LIN {X 0,Y 489.087,Z 544.467,A -85,B 0,C 180,E1 9559.123,E2 9559.123} C_VEL
LIN {X 0,Y 482.604,Z 533.679,A -85,B 0,C 180,E1 9556.552,E2 9556.552} C_VEL
LIN {X 0,Y 477.311,Z 525.25,A -85,B 0,C 180,E1 9554.126,E2 9554.126} C_VEL
LIN {X 0,Y 472.627,Z 517.972,A -85,B 0,C 180,E1 9551.594,E2 9551.594} C_VEL
LIN {X 0,Y 468.762,Z 512.462,A -85,B 0,C 180,E1 9549.082,E2 9549.082} C_VEL
LIN {X 0,Y 465.949,Z 508.396,A -85,B 0,C 180,E1 9546.778,E2 9546.778} C_VEL
LIN {X 0,Y 462.714,Z 503.783,A -85,B 0,C 180,E1 9542.973,E2 9542.973} C_VEL
LIN {X 0,Y 461.058,Z 502.625,A -85,B 0,C 180,E1 9538.633,E2 9538.633} C_VEL
LIN {X 0,Y 461.515,Z 503.464,A -85,B 0,C 180,E1 9534.904,E2 9534.904} C_VEL
LIN {X 0,Y 464.15,Z 508.528,A -85,B 0,C 180,E1 9530.452,E2 9530.452} C_VEL
LIN {X 0,Y 466.705,Z 513.105,A -85,B 0,C 180,E1 9527.943,E2 9527.943} C_VEL
LIN {X 0,Y 469.386,Z 517.69,A -85,B 0,C 180,E1 9525.883,E2 9525.883} C_VEL
LIN {X 0,Y 473.496,Z 524.733,A -85,B 0,C 180,E1 9523.31,E2 9523.31} C_VEL
LIN {X 0,Y 478.239,Z 533.162,A -85,B 0,C 180,E1 9520.837,E2 9520.837} C_VEL
LIN {X 0,Y 483.823,Z 543.406,A -85,B 0,C 180,E1 9518.352,E2 9518.352} C_VEL
LIN {X 0,Y 486.849,Z 549.446,A -85,B 0,C 180,E1 9517.13,E2 9517.13} C_VEL
LIN {X 0,Y 469.793,Z 770.047,A -85,B 0,C 180,E1 9513.766,E2 9513.766} C_VEL
LIN {X 0,Y 464.867,Z 832.514,A -85,B 0,C 180,E1 9512.789,E2 9512.789} C_VEL
LIN {X 0,Y 461.013,Z 860.821,A -85,B 0,C 180,E1 9512.23,E2 9512.23} C_VEL
LIN {X 0,Y 456.896,Z 882.855,A -85,B 0,C 180,E1 9511.67,E2 9511.67} C_VEL
LIN {X 0,Y 452.009,Z 904.689,A -85,B 0,C 180,E1 9510.965,E2 9510.965} C_VEL
LIN {X 0,Y 444.928,Z 930.987,A -85,B 0,C 180,E1 9509.906,E2 9509.906} C_VEL
LIN {X 0,Y 438.503,Z 951.402,A -85,B 0,C 180,E1 9508.895,E2 9508.895} C_VEL
LIN {X 0,Y 431.873,Z 970.249,A -85,B 0,C 180,E1 9507.802,E2 9507.802} C_VEL
LIN {X 0,Y 424.141,Z 990.229,A -85,B 0,C 180,E1 9506.445,E2 9506.445} C_VEL
LIN {X 0,Y 414.213,Z 1013.37,A -85,B 0,C 180,E1 9504.558,E2 9504.558} C_VEL
LIN {X 0,Y 405.888,Z 1031.129,A -85,B 0,C 180,E1 9502.837,E2 9502.837} C_VEL
LIN {X 0,Y 397.662,Z 1047.641,A -85,B 0,C 180,E1 9500.982,E2 9500.982} C_VEL
LIN {X 0,Y 387.672,Z 1066.656,A -85,B 0,C 180,E1 9498.481,E2 9498.481} C_VEL
LIN {X 0,Y 378.087,Z 1083.695,A -85,B 0,C 180,E1 9495.781,E2 9495.781} C_VEL
LIN {X 0,Y 370.336,Z 1097.136,A -85,B 0,C 180,E1 9493.297,E2 9493.297} C_VEL
LIN {X 0,Y 362.061,Z 1111.27,A -85,B 0,C 180,E1 9490.258,E2 9490.258} C_VEL
LIN {X 0,Y 353.591,Z 1125.519,A -85,B 0,C 180,E1 9486.572,E2 9486.572} C_VEL
LIN {X 0,Y 347.43,Z 1136.024,A -85,B 0,C 180,E1 9483.346,E2 9483.346} C_VEL
LIN {X 0,Y 342.159,Z 1145.378,A -85,B 0,C 180,E1 9479.981,E2 9479.981} C_VEL
LIN {X 0,Y 336.708,Z 1155.721,A -85,B 0,C 180,E1 9475.505,E2 9475.505} C_VEL
LIN {X 0,Y 333.16,Z 1163.164,A -85,B 0,C 180,E1 9471.478,E2 9471.478} C_VEL
LIN {X 0,Y 330.879,Z 1168.771,A -85,B 0,C 180,E1 9467.771,E2 9467.771} C_VEL
LIN {X 0,Y 329.229,Z 1173.859,A -85,B 0,C 180,E1 9463.524,E2 9463.524} C_VEL
LIN {X 0,Y 328.351,Z 1177.679,A -85,B 0,C 180,E1 9458.935,E2 9458.935} C_VEL
LIN {X 0,Y 328.063,Z 1179.621,A -85,B 0,C 180,E1 9455.247,E2 9455.247} C_VEL
LIN {X 0,Y 327.994,Z 1180.54,A -85,B 0,C 180,E1 9451.747,E2 9451.747} C_VEL
LIN {X 0,Y 327.999,Z 1180.575,A -85,B 0,C 180,E1 9448.428,E2 9448.428} C_VEL
LIN {X 0,Y 328.045,Z 1179.79,A -85,B 0,C 180,E1 9445.105,E2 9445.105} C_VEL
LIN {X 0,Y 328.254,Z 1178.177,A -85,B 0,C 180,E1 9441.769,E2 9441.769} C_VEL
LIN {X 0,Y 328.768,Z 1175.569,A -85,B 0,C 180,E1 9438.243,E2 9438.243} C_VEL
LIN {X 0,Y 329.903,Z 1171.61,A -85,B 0,C 180,E1 9434.351,E2 9434.351} C_VEL
LIN {X 0,Y 332.358,Z 1165.084,A -85,B 0,C 180,E1 9429.576,E2 9429.576} C_VEL
LIN {X 0,Y 335.423,Z 1158.303,A -85,B 0,C 180,E1 9425.709,E2 9425.709} C_VEL
LIN {X 0,Y 339.344,Z 1150.606,A -85,B 0,C 180,E1 9422.064,E2 9422.064} C_VEL
LIN {X 0,Y 345.374,Z 1139.797,A -85,B 0,C 180,E1 9417.813,E2 9417.813} C_VEL
LIN {X 0,Y 352.237,Z 1127.86,A -85,B 0,C 180,E1 9414.001,E2 9414.001} C_VEL
LIN {X 0,Y 358.846,Z 1116.71,A -85,B 0,C 180,E1 9410.971,E2 9410.971} C_VEL
LIN {X 0,Y 367.61,Z 1102.065,A -85,B 0,C 180,E1 9407.582,E2 9407.582} C_VEL
LIN {X 0,Y 368.215,Z 1100.984,A -85,B 0,C 180,E1 9407.364,E2 9407.364} C_VEL
LIN {X 0,Y 369.925,Z 1096.753,A -85,B 0,C 180,E1 9406.396,E2 9406.396} C_VEL
LIN {X 0,Y 371.745,Z 1086.41,A -85,B 0,C 180,E1 9403.741,E2 9403.741} C_VEL
LIN {X 0,Y 373.805,Z 1081.808,A -85,B 0,C 180,E1 9402.827,E2 9402.827} C_VEL
LIN {X 0,Y 384.889,Z 1062.383,A -85,B 0,C 180,E1 9399.856,E2 9399.856} C_VEL
LIN {X 0,Y 393.525,Z 1046.374,A -85,B 0,C 180,E1 9397.797,E2 9397.797} C_VEL
LIN {X 0,Y 402.328,Z 1029.123,A -85,B 0,C 180,E1 9395.887,E2 9395.887} C_VEL
LIN {X 0,Y 413.045,Z 1006.428,A -85,B 0,C 180,E1 9393.779,E2 9393.779} C_VEL
LIN {X 0,Y 421.336,Z 987.025,A -85,B 0,C 180,E1 9392.273,E2 9392.273} C_VEL
LIN {X 0,Y 428.705,Z 968.221,A -85,B 0,C 180,E1 9391.028,E2 9391.028} C_VEL
LIN {X 0,Y 436.952,Z 944.961,A -85,B 0,C 180,E1 9389.726,E2 9389.726} C_VEL
LIN {X 0,Y 444.264,Z 920.669,A -85,B 0,C 180,E1 9388.629,E2 9388.629} C_VEL
LIN {X 0,Y 449.42,Z 901.022,A -85,B 0,C 180,E1 9387.895,E2 9387.895} C_VEL
LIN {X 0,Y 454.189,Z 879.65,A -85,B 0,C 180,E1 9387.232,E2 9387.232} C_VEL
LIN {X 0,Y 459.09,Z 852.254,A -85,B 0,C 180,E1 9386.579,E2 9386.579} C_VEL
LIN {X 0,Y 462.064,Z 828.163,A -85,B 0,C 180,E1 9386.14,E2 9386.14} C_VEL
LIN {X 0,Y 479.945,Z 602.016,A -85,B 0,C 180,E1 9382.681,E2 9382.681} C_VEL
LIN {X 0,Y 483.792,Z 554.098,A -85,B 0,C 180,E1 9381.936,E2 9381.936} C_VEL
LIN {X 0,Y 478.876,Z 544.784,A -85,B 0,C 180,E1 9379.802,E2 9379.802} C_VEL
LIN {X 0,Y 473.793,Z 535.388,A -85,B 0,C 180,E1 9377.248,E2 9377.248} C_VEL
LIN {X 0,Y 469.705,Z 528.051,A -85,B 0,C 180,E1 9374.8,E2 9374.8} C_VEL
LIN {X 0,Y 466.764,Z 522.997,A -85,B 0,C 180,E1 9372.684,E2 9372.684} C_VEL
LIN {X 0,Y 464.505,Z 518.955,A -85,B 0,C 180,E1 9370.668,E2 9370.668} C_VEL
LIN {X 0,Y 462.693,Z 515.548,A -85,B 0,C 180,E1 9368.575,E2 9368.575} C_VEL
LIN {X 0,Y 460.581,Z 511.278,A -85,B 0,C 180,E1 9364.233,E2 9364.233} C_VEL
LIN {X 0,Y 460.586,Z 510.886,A -85,B 0,C 180,E1 9360.124,E2 9360.124} C_VEL
LIN {X 0,Y 462.046,Z 512.115,A -85,B 0,C 180,E1 9356.899,E2 9356.899} C_VEL
LIN {X 0,Y 465.598,Z 517.283,A -85,B 0,C 180,E1 9352.813,E2 9352.813} C_VEL
LIN {X 0,Y 468.807,Z 522.051,A -85,B 0,C 180,E1 9350.3,E2 9350.3} C_VEL
LIN {X 0,Y 472.497,Z 527.678,A -85,B 0,C 180,E1 9347.969,E2 9347.969} C_VEL
LIN {X 0,Y 476.763,Z 534.255,A -85,B 0,C 180,E1 9345.703,E2 9345.703} C_VEL
LIN {X 0,Y 482.388,Z 543.628,A -85,B 0,C 180,E1 9343.131,E2 9343.131} C_VEL
LIN {X 0,Y 485.974,Z 549.849,A -85,B 0,C 180,E1 9341.67,E2 9341.67} C_VEL
LIN {X 0,Y 467.737,Z 771.285,A -85,B 0,C 180,E1 9338.178,E2 9338.178} C_VEL
LIN {X 0,Y 462.75,Z 830.028,A -85,B 0,C 180,E1 9337.224,E2 9337.224} C_VEL
LIN {X 0,Y 458.58,Z 859.423,A -85,B 0,C 180,E1 9336.635,E2 9336.635} C_VEL
LIN {X 0,Y 454.315,Z 881.758,A -85,B 0,C 180,E1 9336.059,E2 9336.059} C_VEL
LIN {X 0,Y 449.542,Z 902.729,A -85,B 0,C 180,E1 9335.387,E2 9335.387} C_VEL
LIN {X 0,Y 443.382,Z 925.948,A -85,B 0,C 180,E1 9334.486,E2 9334.486} C_VEL
LIN {X 0,Y 435.171,Z 952.253,A -85,B 0,C 180,E1 9333.221,E2 9333.221} C_VEL
LIN {X 0,Y 427.918,Z 972.779,A -85,B 0,C 180,E1 9332.035,E2 9332.035} C_VEL
LIN {X 0,Y 420.219,Z 992.621,A -85,B 0,C 180,E1 9330.695,E2 9330.695} C_VEL
LIN {X 0,Y 410.557,Z 1015.499,A -85,B 0,C 180,E1 9328.875,E2 9328.875} C_VEL
LIN {X 0,Y 400.827,Z 1036.337,A -85,B 0,C 180,E1 9326.886,E2 9326.886} C_VEL
LIN {X 0,Y 392.615,Z 1052.989,A -85,B 0,C 180,E1 9325.039,E2 9325.039} C_VEL
LIN {X 0,Y 384.33,Z 1068.988,A -85,B 0,C 180,E1 9323.005,E2 9323.005} C_VEL
LIN {X 0,Y 374.751,Z 1086.828,A -85,B 0,C 180,E1 9320.38,E2 9320.38} C_VEL
LIN {X 0,Y 364.261,Z 1105.498,A -85,B 0,C 180,E1 9317.097,E2 9317.097} C_VEL
LIN {X 0,Y 356.529,Z 1119.082,A -85,B 0,C 180,E1 9314.291,E2 9314.291} C_VEL
LIN {X 0,Y 349.143,Z 1132.063,A -85,B 0,C 180,E1 9311.198,E2 9311.198} C_VEL
LIN {X 0,Y 341.061,Z 1146.648,A -85,B 0,C 180,E1 9307.115,E2 9307.115} C_VEL
LIN {X 0,Y 334.709,Z 1158.415,A -85,B 0,C 180,E1 9303.139,E2 9303.139} C_VEL
LIN {X 0,Y 330.228,Z 1167.436,A -85,B 0,C 180,E1 9299.573,E2 9299.573} C_VEL
LIN {X 0,Y 326.523,Z 1175.647,A -85,B 0,C 180,E1 9295.774,E2 9295.774} C_VEL
LIN {X 0,Y 323.261,Z 1184.188,A -85,B 0,C 180,E1 9291.026,E2 9291.026} C_VEL
LIN {X 0,Y 321.327,Z 1190.525,A -85,B 0,C 180,E1 9286.449,E2 9286.449} C_VEL
LIN {X 0,Y 320.465,Z 1194.51,A -85,B 0,C 180,E1 9282.798,E2 9282.798} C_VEL
LIN {X 0,Y 320.083,Z 1197.498,A -85,B 0,C 180,E1 9279.167,E2 9279.167} C_VEL
LIN {X 0,Y 319.974,Z 1199.429,A -85,B 0,C 180,E1 9275.739,E2 9275.739} C_VEL
LIN {X 0,Y 319.968,Z 1200.477,A -85,B 0,C 180,E1 9272.328,E2 9272.328} C_VEL
LIN {X 0,Y 319.971,Z 1200.644,A -85,B 0,C 180,E1 9268.925,E2 9268.925} C_VEL
LIN {X 0,Y 319.965,Z 1199.856,A -85,B 0,C 180,E1 9265.339,E2 9265.339} C_VEL
LIN {X 0,Y 320.041,Z 1198.091,A -85,B 0,C 180,E1 9261.737,E2 9261.737} C_VEL
LIN {X 0,Y 320.327,Z 1195.341,A -85,B 0,C 180,E1 9258.111,E2 9258.111} C_VEL
LIN {X 0,Y 321.061,Z 1191.597,A -85,B 0,C 180,E1 9254.464,E2 9254.464} C_VEL
LIN {X 0,Y 322.419,Z 1186.569,A -85,B 0,C 180,E1 9250.62,E2 9250.62} C_VEL
LIN {X 0,Y 324.462,Z 1180.714,A -85,B 0,C 180,E1 9246.96,E2 9246.96} C_VEL
LIN {X 0,Y 327.643,Z 1173.043,A -85,B 0,C 180,E1 9242.954,E2 9242.954} C_VEL
LIN {X 0,Y 333.044,Z 1161.711,A -85,B 0,C 180,E1 9238.103,E2 9238.103} C_VEL
LIN {X 0,Y 338.43,Z 1151.31,A -85,B 0,C 180,E1 9234.406,E2 9234.406} C_VEL
LIN {X 0,Y 344.378,Z 1140.469,A -85,B 0,C 180,E1 9231.09,E2 9231.09} C_VEL
LIN {X 0,Y 351.395,Z 1128.08,A -85,B 0,C 180,E1 9227.815,E2 9227.815} C_VEL
LIN {X 0,Y 361.198,Z 1110.841,A -85,B 0,C 180,E1 9223.967,E2 9223.967} C_VEL
LIN {X 0,Y 369.441,Z 1096.146,A -85,B 0,C 180,E1 9221.201,E2 9221.201} C_VEL
LIN {X 0,Y 377.651,Z 1081.262,A -85,B 0,C 180,E1 9218.773,E2 9218.773} C_VEL
LIN {X 0,Y 386.777,Z 1064.204,A -85,B 0,C 180,E1 9216.363,E2 9216.363} C_VEL
LIN {X 0,Y 397.957,Z 1042.084,A -85,B 0,C 180,E1 9213.73,E2 9213.73} C_VEL
LIN {X 0,Y 406.908,Z 1023.145,A -85,B 0,C 180,E1 9211.835,E2 9211.835} C_VEL
LIN {X 0,Y 415.23,Z 1004.37,A -85,B 0,C 180,E1 9210.217,E2 9210.217} C_VEL
LIN {X 0,Y 424.56,Z 981.647,A -85,B 0,C 180,E1 9208.544,E2 9208.544} C_VEL
LIN {X 0,Y 433.034,Z 958.176,A -85,B 0,C 180,E1 9207.111,E2 9207.111} C_VEL
LIN {X 0,Y 439.667,Z 937.838,A -85,B 0,C 180,E1 9206.064,E2 9206.064} C_VEL
LIN {X 0,Y 445.723,Z 916.98,A -85,B 0,C 180,E1 9205.155,E2 9205.155} C_VEL
LIN {X 0,Y 452.319,Z 890.732,A -85,B 0,C 180,E1 9204.217,E2 9204.217} C_VEL
LIN {X 0,Y 457.368,Z 865.454,A -85,B 0,C 180,E1 9203.515,E2 9203.515} C_VEL
LIN {X 0,Y 460.917,Z 843.374,A -85,B 0,C 180,E1 9203.034,E2 9203.034} C_VEL
LIN {X 0,Y 463.734,Z 818.818,A -85,B 0,C 180,E1 9202.591,E2 9202.591} C_VEL
LIN {X 0,Y 481.973,Z 595.843,A -85,B 0,C 180,E1 9199.059,E2 9199.059} C_VEL
LIN {X 0,Y 485.822,Z 549.536,A -85,B 0,C 180,E1 9198.324,E2 9198.324} C_VEL
LIN {X 0,Y 478.853,Z 537.763,A -85,B 0,C 180,E1 9195.378,E2 9195.378} C_VEL
LIN {X 0,Y 473.264,Z 528.913,A -85,B 0,C 180,E1 9192.569,E2 9192.569} C_VEL
LIN {X 0,Y 470.141,Z 524.264,A -85,B 0,C 180,E1 9190.725,E2 9190.725} C_VEL
LIN {X 0,Y 467.433,Z 520.15,A -85,B 0,C 180,E1 9188.86,E2 9188.86} C_VEL
LIN {X 0,Y 464.829,Z 516.268,A -85,B 0,C 180,E1 9186.671,E2 9186.671} C_VEL
LIN {X 0,Y 461.652,Z 511.681,A -85,B 0,C 180,E1 9182.855,E2 9182.855} C_VEL
LIN {X 0,Y 460.081,Z 510.564,A -85,B 0,C 180,E1 9178.607,E2 9178.607} C_VEL
LIN {X 0,Y 460.501,Z 511.348,A -85,B 0,C 180,E1 9175.017,E2 9175.017} C_VEL
LIN {X 0,Y 463.017,Z 516.34,A -85,B 0,C 180,E1 9170.616,E2 9170.616} C_VEL
LIN {X 0,Y 465.518,Z 520.942,A -85,B 0,C 180,E1 9168.1,E2 9168.1} C_VEL
LIN {X 0,Y 468.15,Z 525.563,A -85,B 0,C 180,E1 9166.034,E2 9166.034} C_VEL
LIN {X 0,Y 471.989,Z 532.31,A -85,B 0,C 180,E1 9163.572,E2 9163.572} C_VEL
LIN {X 0,Y 476.548,Z 540.594,A -85,B 0,C 180,E1 9161.134,E2 9161.134} C_VEL
LIN {X 0,Y 481.912,Z 550.674,A -85,B 0,C 180,E1 9158.685,E2 9158.685} C_VEL
LIN {X 0,Y 483.658,Z 554.297,A -85,B 0,C 180,E1 9157.946,E2 9157.946} C_VEL
LIN {X 0,Y 466.085,Z 776.087,A -85,B 0,C 180,E1 9154.572,E2 9154.572} C_VEL
LIN {X 0,Y 461.441,Z 833.039,A -85,B 0,C 180,E1 9153.681,E2 9153.681} C_VEL
LIN {X 0,Y 457.508,Z 861.097,A -85,B 0,C 180,E1 9153.129,E2 9153.129} C_VEL
LIN {X 0,Y 453.293,Z 883.182,A -85,B 0,C 180,E1 9152.571,E2 9152.571} C_VEL
LIN {X 0,Y 448.197,Z 905.439,A -85,B 0,C 180,E1 9151.856,E2 9151.856} C_VEL
LIN {X 0,Y 440.972,Z 931.565,A -85,B 0,C 180,E1 9150.805,E2 9150.805} C_VEL
LIN {X 0,Y 434.412,Z 951.92,A -85,B 0,C 180,E1 9149.801,E2 9149.801} C_VEL
LIN {X 0,Y 427.637,Z 970.722,A -85,B 0,C 180,E1 9148.715,E2 9148.715} C_VEL
LIN {X 0,Y 419.173,Z 992.057,A -85,B 0,C 180,E1 9147.262,E2 9147.262} C_VEL
LIN {X 0,Y 409.25,Z 1014.406,A -85,B 0,C 180,E1 9145.423,E2 9145.423} C_VEL
LIN {X 0,Y 400.725,Z 1032.084,A -85,B 0,C 180,E1 9143.702,E2 9143.702} C_VEL
LIN {X 0,Y 392.007,Z 1049.072,A -85,B 0,C 180,E1 9141.777,E2 9141.777} C_VEL
LIN {X 0,Y 381.06,Z 1069.057,A -85,B 0,C 180,E1 9139.086,E2 9139.086} C_VEL
LIN {X 0,Y 372.4,Z 1083.999,A -85,B 0,C 180,E1 9136.688,E2 9136.688} C_VEL
LIN {X 0,Y 363.931,Z 1098.184,A -85,B 0,C 180,E1 9134.036,E2 9134.036} C_VEL
LIN {X 0,Y 354.599,Z 1113.556,A -85,B 0,C 180,E1 9130.645,E2 9130.645} C_VEL
LIN {X 0,Y 346.39,Z 1126.747,A -85,B 0,C 180,E1 9127.106,E2 9127.106} C_VEL
LIN {X 0,Y 339.955,Z 1137.294,A -85,B 0,C 180,E1 9123.772,E2 9123.772} C_VEL
LIN {X 0,Y 333.509,Z 1148.386,A -85,B 0,C 180,E1 9119.605,E2 9119.605} C_VEL
LIN {X 0,Y 328.4,Z 1157.61,A -85,B 0,C 180,E1 9115.272,E2 9115.272} C_VEL
LIN {X 0,Y 325.124,Z 1164.296,A -85,B 0,C 180,E1 9111.468,E2 9111.468} C_VEL
LIN {X 0,Y 322.483,Z 1170.734,A -85,B 0,C 180,E1 9106.945,E2 9106.945} C_VEL
LIN {X 0,Y 320.934,Z 1175.425,A -85,B 0,C 180,E1 9102.414,E2 9102.414} C_VEL
LIN {X 0,Y 320.322,Z 1178.252,A -85,B 0,C 180,E1 9098.618,E2 9098.618} C_VEL
LIN {X 0,Y 320.057,Z 1179.998,A -85,B 0,C 180,E1 9095.019,E2 9095.019} C_VEL
LIN {X 0,Y 319.997,Z 1180.809,A -85,B 0,C 180,E1 9091.612,E2 9091.612} C_VEL
LIN {X 0,Y 320.006,Z 1180.8,A -85,B 0,C 180,E1 9088.21,E2 9088.21} C_VEL
LIN {X 0,Y 320.062,Z 1179.973,A -85,B 0,C 180,E1 9084.802,E2 9084.802} C_VEL
LIN {X 0,Y 320.332,Z 1178.21,A -85,B 0,C 180,E1 9081.203,E2 9081.203} C_VEL
LIN {X 0,Y 321.004,Z 1175.212,A -85,B 0,C 180,E1 9077.224,E2 9077.224} C_VEL
LIN {X 0,Y 322.785,Z 1169.902,A -85,B 0,C 180,E1 9072.328,E2 9072.328} C_VEL
LIN {X 0,Y 325.195,Z 1164.177,A -85,B 0,C 180,E1 9068.349,E2 9068.349} C_VEL
LIN {X 0,Y 328.462,Z 1157.543,A -85,B 0,C 180,E1 9064.582,E2 9064.582} C_VEL
LIN {X 0,Y 333.698,Z 1148.116,A -85,B 0,C 180,E1 9060.173,E2 9060.173} C_VEL
LIN {X 0,Y 340.123,Z 1137.072,A -85,B 0,C 180,E1 9056.045,E2 9056.045} C_VEL
LIN {X 0,Y 346.595,Z 1126.496,A -85,B 0,C 180,E1 9052.713,E2 9052.713} C_VEL
LIN {X 0,Y 355.244,Z 1112.617,A -85,B 0,C 180,E1 9049.02,E2 9049.02} C_VEL
LIN {X 0,Y 364.316,Z 1097.665,A -85,B 0,C 180,E1 9045.753,E2 9045.753} C_VEL
LIN {X 0,Y 372.539,Z 1083.908,A -85,B 0,C 180,E1 9043.19,E2 9043.19} C_VEL
LIN {X 0,Y 373.805,Z 1081.808,A -85,B 0,C 180,E1 9042.827,E2 9042.827} C_VEL
LIN {X 0,Y 375.924,Z 1077.178,A -85,B 0,C 180,E1 9041.932,E2 9041.932} C_VEL
LIN {X 0,Y 378.862,Z 1065.068,A -85,B 0,C 180,E1 9039.326,E2 9039.326} C_VEL
LIN {X 0,Y 380.839,Z 1060.662,A -85,B 0,C 180,E1 9038.629,E2 9038.629} C_VEL
LIN {X 0,Y 389.359,Z 1045.266,A -85,B 0,C 180,E1 9036.675,E2 9036.675} C_VEL
LIN {X 0,Y 398.942,Z 1026.928,A -85,B 0,C 180,E1 9034.677,E2 9034.677} C_VEL
LIN {X 0,Y 409.366,Z 1005.103,A -85,B 0,C 180,E1 9032.695,E2 9032.695} C_VEL
LIN {X 0,Y 417.191,Z 987.19,A -85,B 0,C 180,E1 9031.318,E2 9031.318} C_VEL
LIN {X 0,Y 424.767,Z 968.28,A -85,B 0,C 180,E1 9030.072,E2 9030.072} C_VEL
LIN {X 0,Y 433.029,Z 945.469,A -85,B 0,C 180,E1 9028.804,E2 9028.804} C_VEL
LIN {X 0,Y 440.491,Z 921.305,A -85,B 0,C 180,E1 9027.716,E2 9027.716} C_VEL
LIN {X 0,Y 445.748,Z 901.755,A -85,B 0,C 180,E1 9026.99,E2 9026.99} C_VEL
LIN {X 0,Y 450.512,Z 880.944,A -85,B 0,C 180,E1 9026.344,E2 9026.344} C_VEL
LIN {X 0,Y 455.419,Z 854.865,A -85,B 0,C 180,E1 9025.713,E2 9025.713} C_VEL
LIN {X 0,Y 458.75,Z 828.848,A -85,B 0,C 180,E1 9025.237,E2 9025.237} C_VEL
LIN {X 0,Y 477.095,Z 602.943,A -85,B 0,C 180,E1 9021.793,E2 9021.793} C_VEL
LIN {X 0,Y 480.703,Z 559.088,A -85,B 0,C 180,E1 9021.112,E2 9021.112} C_VEL
LIN {X 0,Y 475.753,Z 549.457,A -85,B 0,C 180,E1 9018.821,E2 9018.821} C_VEL
LIN {X 0,Y 471.327,Z 541.288,A -85,B 0,C 180,E1 9016.452,E2 9016.452} C_VEL
LIN {X 0,Y 467.998,Z 535.179,A -85,B 0,C 180,E1 9014.35,E2 9014.35} C_VEL
LIN {X 0,Y 465.483,Z 530.695,A -85,B 0,C 180,E1 9012.467,E2 9012.467} C_VEL
LIN {X 0,Y 463.167,Z 526.461,A -85,B 0,C 180,E1 9010.322,E2 9010.322} C_VEL
LIN {X 0,Y 461.534,Z 523.318,A -85,B 0,C 180,E1 9008.346,E2 9008.346} C_VEL
LIN {X 0,Y 459.608,Z 519.226,A -85,B 0,C 180,E1 9004.242,E2 9004.242} C_VEL
LIN {X 0,Y 459.58,Z 518.808,A -85,B 0,C 180,E1 9000.249,E2 9000.249} C_VEL
LIN {X 0,Y 461.055,Z 520.15,A -85,B 0,C 180,E1 8996.892,E2 8996.892} C_VEL
LIN {X 0,Y 464.429,Z 525.143,A -85,B 0,C 180,E1 8992.951,E2 8992.951} C_VEL
LIN {X 0,Y 467.545,Z 529.883,A -85,B 0,C 180,E1 8990.46,E2 8990.46} C_VEL
LIN {X 0,Y 470.977,Z 535.209,A -85,B 0,C 180,E1 8988.24,E2 8988.24} C_VEL
LIN {X 0,Y 475.148,Z 541.808,A -85,B 0,C 180,E1 8985.964,E2 8985.964} C_VEL
LIN {X 0,Y 480.604,Z 551.1,A -85,B 0,C 180,E1 8983.408,E2 8983.408} C_VEL
LIN {X 0,Y 482.79,Z 555.033,A -85,B 0,C 180,E1 8982.482,E2 8982.482} C_VEL
LIN {X 0,Y 464.15,Z 776.331,A -85,B 0,C 180,E1 8979.005,E2 8979.005} C_VEL
LIN {X 0,Y 459.389,Z 830.749,A -85,B 0,C 180,E1 8978.122,E2 8978.122} C_VEL
LIN {X 0,Y 455.185,Z 859.62,A -85,B 0,C 180,E1 8977.546,E2 8977.546} C_VEL
LIN {X 0,Y 450.857,Z 881.859,A -85,B 0,C 180,E1 8976.977,E2 8976.977} C_VEL
LIN {X 0,Y 445.848,Z 903.395,A -85,B 0,C 180,E1 8976.292,E2 8976.292} C_VEL
LIN {X 0,Y 439.052,Z 928.394,A -85,B 0,C 180,E1 8975.321,E2 8975.321} C_VEL
LIN {X 0,Y 431.135,Z 952.846,A -85,B 0,C 180,E1 8974.136,E2 8974.136} C_VEL
LIN {X 0,Y 423.86,Z 972.947,A -85,B 0,C 180,E1 8972.98,E2 8972.98} C_VEL
LIN {X 0,Y 415.898,Z 992.984,A -85,B 0,C 180,E1 8971.631,E2 8971.631} C_VEL
LIN {X 0,Y 405.668,Z 1016.473,A -85,B 0,C 180,E1 8969.757,E2 8969.757} C_VEL
LIN {X 0,Y 395.819,Z 1036.987,A -85,B 0,C 180,E1 8967.791,E2 8967.791} C_VEL
LIN {X 0,Y 387.347,Z 1053.65,A -85,B 0,C 180,E1 8965.933,E2 8965.933} C_VEL
LIN {X 0,Y 378.44,Z 1070.303,A -85,B 0,C 180,E1 8963.795,E2 8963.795} C_VEL
LIN {X 0,Y 367.511,Z 1089.864,A -85,B 0,C 180,E1 8960.84,E2 8960.84} C_VEL
LIN {X 0,Y 358.041,Z 1106.068,A -85,B 0,C 180,E1 8957.914,E2 8957.914} C_VEL
LIN {X 0,Y 350.099,Z 1119.505,A -85,B 0,C 180,E1 8955.095,E2 8955.095} C_VEL
LIN {X 0,Y 342.062,Z 1133.078,A -85,B 0,C 180,E1 8951.794,E2 8951.794} C_VEL
LIN {X 0,Y 333.141,Z 1148.406,A -85,B 0,C 180,E1 8947.32,E2 8947.32} C_VEL
LIN {X 0,Y 327.417,Z 1158.614,A -85,B 0,C 180,E1 8943.765,E2 8943.765} C_VEL
LIN {X 0,Y 322.731,Z 1167.585,A -85,B 0,C 180,E1 8940.126,E2 8940.126} C_VEL
LIN {X 0,Y 318.692,Z 1176.115,A -85,B 0,C 180,E1 8936.055,E2 8936.055} C_VEL
LIN {X 0,Y 315.112,Z 1184.993,A -85,B 0,C 180,E1 8930.817,E2 8930.817} C_VEL
LIN {X 0,Y 313.388,Z 1190.485,A -85,B 0,C 180,E1 8926.687,E2 8926.687} C_VEL
LIN {X 0,Y 312.484,Z 1194.425,A -85,B 0,C 180,E1 8922.943,E2 8922.943} C_VEL
LIN {X 0,Y 312.093,Z 1197.297,A -85,B 0,C 180,E1 8919.326,E2 8919.326} C_VEL
LIN {X 0,Y 311.977,Z 1199.18,A -85,B 0,C 180,E1 8915.886,E2 8915.886} C_VEL
LIN {X 0,Y 311.971,Z 1200.23,A -85,B 0,C 180,E1 8912.388,E2 8912.388} C_VEL
LIN {X 0,Y 311.975,Z 1200.397,A -85,B 0,C 180,E1 8908.898,E2 8908.898} C_VEL
LIN {X 0,Y 311.969,Z 1199.608,A -85,B 0,C 180,E1 8905.22,E2 8905.22} C_VEL
LIN {X 0,Y 312.049,Z 1197.84,A -85,B 0,C 180,E1 8901.524,E2 8901.524} C_VEL
LIN {X 0,Y 312.368,Z 1195.087,A -85,B 0,C 180,E1 8897.803,E2 8897.803} C_VEL
LIN {X 0,Y 313.162,Z 1191.339,A -85,B 0,C 180,E1 8894.062,E2 8894.062} C_VEL
LIN {X 0,Y 314.595,Z 1186.399,A -85,B 0,C 180,E1 8890.185,E2 8890.185} C_VEL
LIN {X 0,Y 316.816,Z 1180.448,A -85,B 0,C 180,E1 8886.371,E2 8886.371} C_VEL
LIN {X 0,Y 320.383,Z 1172.405,A -85,B 0,C 180,E1 8882.086,E2 8882.086} C_VEL
LIN {X 0,Y 326.157,Z 1160.955,A -85,B 0,C 180,E1 8877.138,E2 8877.138} C_VEL
LIN {X 0,Y 331.9,Z 1150.493,A -85,B 0,C 180,E1 8873.38,E2 8873.38} C_VEL
LIN {X 0,Y 338.363,Z 1139.315,A -85,B 0,C 180,E1 8869.94,E2 8869.94} C_VEL
LIN {X 0,Y 347.169,Z 1124.474,A -85,B 0,C 180,E1 8866.044,E2 8866.044} C_VEL
LIN {X 0,Y 356.28,Z 1108.946,A -85,B 0,C 180,E1 8862.668,E2 8862.668} C_VEL
LIN {X 0,Y 364.431,Z 1094.959,A -85,B 0,C 180,E1 8860.05,E2 8860.05} C_VEL
LIN {X 0,Y 373.255,Z 1079.477,A -85,B 0,C 180,E1 8857.54,E2 8857.54} C_VEL
LIN {X 0,Y 384.164,Z 1059.637,A -85,B 0,C 180,E1 8854.798,E2 8854.798} C_VEL
LIN {X 0,Y 394.283,Z 1039.864,A -85,B 0,C 180,E1 8852.522,E2 8852.522} C_VEL
LIN {X 0,Y 403.035,Z 1021.759,A -85,B 0,C 180,E1 8850.735,E2 8850.735} C_VEL
LIN {X 0,Y 412.535,Z 1000.739,A -85,B 0,C 180,E1 8848.958,E2 8848.958} C_VEL
LIN {X 0,Y 422.368,Z 976.596,A -85,B 0,C 180,E1 8847.261,E2 8847.261} C_VEL
LIN {X 0,Y 429.696,Z 956.617,A -85,B 0,C 180,E1 8846.077,E2 8846.077} C_VEL
LIN {X 0,Y 436.122,Z 937.241,A -85,B 0,C 180,E1 8845.095,E2 8845.095} C_VEL
LIN {X 0,Y 442.674,Z 915.012,A -85,B 0,C 180,E1 8844.143,E2 8844.143} C_VEL
LIN {X 0,Y 449.683,Z 886.727,A -85,B 0,C 180,E1 8843.174,E2 8843.174} C_VEL
LIN {X 0,Y 454.204,Z 864.236,A -85,B 0,C 180,E1 8842.569,E2 8842.569} C_VEL
LIN {X 0,Y 457.768,Z 842.166,A -85,B 0,C 180,E1 8842.099,E2 8842.099} C_VEL
LIN {X 0,Y 460.875,Z 814.57,A -85,B 0,C 180,E1 8841.61,E2 8841.61} C_VEL
LIN {X 0,Y 479.731,Z 588.85,A -85,B 0,C 180,E1 8838.053,E2 8838.053} C_VEL
LIN {X 0,Y 482.639,Z 554.74,A -85,B 0,C 180,E1 8837.517,E2 8837.517} C_VEL
LIN {X 0,Y 476.697,Z 544.545,A -85,B 0,C 180,E1 8834.889,E2 8834.889} C_VEL
LIN {X 0,Y 471.612,Z 536.292,A -85,B 0,C 180,E1 8832.241,E2 8832.241} C_VEL
LIN {X 0,Y 468.577,Z 531.674,A -85,B 0,C 180,E1 8830.388,E2 8830.388} C_VEL
LIN {X 0,Y 466.113,Z 527.837,A -85,B 0,C 180,E1 8828.636,E2 8828.636} C_VEL
LIN {X 0,Y 463.577,Z 524.003,A -85,B 0,C 180,E1 8826.44,E2 8826.44} C_VEL
LIN {X 0,Y 460.591,Z 519.579,A -85,B 0,C 180,E1 8822.737,E2 8822.737} C_VEL
LIN {X 0,Y 459.097,Z 518.501,A -85,B 0,C 180,E1 8818.502,E2 8818.502} C_VEL
LIN {X 0,Y 459.52,Z 519.366,A -85,B 0,C 180,E1 8815.007,E2 8815.007} C_VEL
LIN {X 0,Y 461.887,Z 524.151,A -85,B 0,C 180,E1 8810.782,E2 8810.782} C_VEL
LIN {X 0,Y 464.328,Z 528.776,A -85,B 0,C 180,E1 8808.258,E2 8808.258} C_VEL
LIN {X 0,Y 466.753,Z 533.117,A -85,B 0,C 180,E1 8806.307,E2 8806.307} C_VEL
LIN {X 0,Y 470.429,Z 539.755,A -85,B 0,C 180,E1 8803.874,E2 8803.874} C_VEL
LIN {X 0,Y 474.879,Z 548.036,A -85,B 0,C 180,E1 8801.43,E2 8801.43} C_VEL
LIN {X 0,Y 479.982,Z 557.868,A -85,B 0,C 180,E1 8799.036,E2 8799.036} C_VEL
LIN {X 0,Y 480.559,Z 559.318,A -85,B 0,C 180,E1 8798.77,E2 8798.77} C_VEL
LIN {X 0,Y 462.56,Z 781.004,A -85,B 0,C 180,E1 8795.409,E2 8795.409} C_VEL
LIN {X 0,Y 458.095,Z 833.883,A -85,B 0,C 180,E1 8794.581,E2 8794.581} C_VEL
LIN {X 0,Y 454.115,Z 861.388,A -85,B 0,C 180,E1 8794.04,E2 8794.04} C_VEL
LIN {X 0,Y 449.827,Z 883.404,A -85,B 0,C 180,E1 8793.489,E2 8793.489} C_VEL
LIN {X 0,Y 444.677,Z 905.455,A -85,B 0,C 180,E1 8792.786,E2 8792.786} C_VEL
LIN {X 0,Y 437.126,Z 932.142,A -85,B 0,C 180,E1 8791.721,E2 8791.721} C_VEL
LIN {X 0,Y 430.432,Z 952.438,A -85,B 0,C 180,E1 8790.724,E2 8790.724} C_VEL
LIN {X 0,Y 423.589,Z 970.993,A -85,B 0,C 180,E1 8789.658,E2 8789.658} C_VEL
LIN {X 0,Y 414.734,Z 992.801,A -85,B 0,C 180,E1 8788.178,E2 8788.178} C_VEL
LIN {X 0,Y 404.702,Z 1014.784,A -85,B 0,C 180,E1 8786.368,E2 8786.368} C_VEL
LIN {X 0,Y 395.964,Z 1032.443,A -85,B 0,C 180,E1 8784.65,E2 8784.65} C_VEL
LIN {X 0,Y 386.728,Z 1049.944,A -85,B 0,C 180,E1 8782.662,E2 8782.662} C_VEL
LIN {X 0,Y 375.198,Z 1070.276,A -85,B 0,C 180,E1 8779.893,E2 8779.893} C_VEL
LIN {X 0,Y 366.304,Z 1085.131,A -85,B 0,C 180,E1 8777.477,E2 8777.477} C_VEL
LIN {X 0,Y 357.13,Z 1099.986,A -85,B 0,C 180,E1 8774.648,E2 8774.648} C_VEL
LIN {X 0,Y 346.895,Z 1116.053,A -85,B 0,C 180,E1 8770.958,E2 8770.958} C_VEL
LIN {X 0,Y 339.473,Z 1127.582,A -85,B 0,C 180,E1 8767.781,E2 8767.781} C_VEL
LIN {X 0,Y 332.805,Z 1138.067,A -85,B 0,C 180,E1 8764.391,E2 8764.391} C_VEL
LIN {X 0,Y 325.66,Z 1149.736,A -85,B 0,C 180,E1 8759.828,E2 8759.828} C_VEL
LIN {X 0,Y 320.804,Z 1158.17,A -85,B 0,C 180,E1 8755.741,E2 8755.741} C_VEL
LIN {X 0,Y 317.36,Z 1164.848,A -85,B 0,C 180,E1 8751.825,E2 8751.825} C_VEL
LIN {X 0,Y 314.506,Z 1171.411,A -85,B 0,C 180,E1 8747.007,E2 8747.007} C_VEL
LIN {X 0,Y 312.972,Z 1175.828,A -85,B 0,C 180,E1 8742.548,E2 8742.548} C_VEL
LIN {X 0,Y 312.332,Z 1178.609,A -85,B 0,C 180,E1 8738.654,E2 8738.654} C_VEL
LIN {X 0,Y 312.06,Z 1180.311,A -85,B 0,C 180,E1 8734.963,E2 8734.963} C_VEL
LIN {X 0,Y 312.003,Z 1181.099,A -85,B 0,C 180,E1 8731.286,E2 8731.286} C_VEL
LIN {X 0,Y 312.012,Z 1180.984,A -85,B 0,C 180,E1 8727.613,E2 8727.613} C_VEL
LIN {X 0,Y 312.161,Z 1179.709,A -85,B 0,C 180,E1 8723.194,E2 8723.194} C_VEL
LIN {X 0,Y 312.715,Z 1176.831,A -85,B 0,C 180,E1 8718.566,E2 8718.566} C_VEL
LIN {X 0,Y 313.86,Z 1173.103,A -85,B 0,C 180,E1 8714.479,E2 8714.479} C_VEL
LIN {X 0,Y 315.708,Z 1168.452,A -85,B 0,C 180,E1 8710.577,E2 8710.577} C_VEL
LIN {X 0,Y 319.102,Z 1161.523,A -85,B 0,C 180,E1 8705.962,E2 8705.962} C_VEL
LIN {X 0,Y 323.928,Z 1152.697,A -85,B 0,C 180,E1 8701.417,E2 8701.417} C_VEL
LIN {X 0,Y 328.901,Z 1144.386,A -85,B 0,C 180,E1 8697.859,E2 8697.859} C_VEL
LIN {X 0,Y 335.563,Z 1133.842,A -85,B 0,C 180,E1 8694.056,E2 8694.056} C_VEL
LIN {X 0,Y 344.183,Z 1120.358,A -85,B 0,C 180,E1 8690.058,E2 8690.058} C_VEL
LIN {X 0,Y 352.022,Z 1108.116,A -85,B 0,C 180,E1 8687.025,E2 8687.025} C_VEL
LIN {X 0,Y 360.246,Z 1095.118,A -85,B 0,C 180,E1 8684.268,E2 8684.268} C_VEL
LIN {X 0,Y 370.775,Z 1078.016,A -85,B 0,C 180,E1 8681.203,E2 8681.203} C_VEL
LIN {X 0,Y 380.839,Z 1060.662,A -85,B 0,C 180,E1 8678.629,E2 8678.629} C_VEL
LIN {X 0,Y 383.13,Z 1055.589,A -85,B 0,C 180,E1 8677.819,E2 8677.819} C_VEL
LIN {X 0,Y 386.851,Z 1042.392,A -85,B 0,C 180,E1 8675.402,E2 8675.402} C_VEL
LIN {X 0,Y 388.916,Z 1037.652,A -85,B 0,C 180,E1 8674.785,E2 8674.785} C_VEL
LIN {X 0,Y 398.767,Z 1018.463,A -85,B 0,C 180,E1 8672.862,E2 8672.862} C_VEL
LIN {X 0,Y 407.34,Z 1000.495,A -85,B 0,C 180,E1 8671.327,E2 8671.327} C_VEL
LIN {X 0,Y 416.662,Z 979.252,A -85,B 0,C 180,E1 8669.785,E2 8669.785} C_VEL
LIN {X 0,Y 425.654,Z 955.915,A -85,B 0,C 180,E1 8668.393,E2 8668.393} C_VEL
LIN {X 0,Y 432.091,Z 937.166,A -85,B 0,C 180,E1 8667.448,E2 8667.448} C_VEL
LIN {X 0,Y 438.286,Z 916.844,A -85,B 0,C 180,E1 8666.584,E2 8666.584} C_VEL
LIN {X 0,Y 444.795,Z 892.188,A -85,B 0,C 180,E1 8665.729,E2 8665.729} C_VEL
LIN {X 0,Y 450.121,Z 866.522,A -85,B 0,C 180,E1 8665.047,E2 8665.047} C_VEL
LIN {X 0,Y 453.639,Z 844.978,A -85,B 0,C 180,E1 8664.596,E2 8664.596} C_VEL
LIN {X 0,Y 456.508,Z 820.105,A -85,B 0,C 180,E1 8664.168,E2 8664.168} C_VEL
LIN {X 0,Y 475.434,Z 591.235,A -85,B 0,C 180,E1 8660.702,E2 8660.702} C_VEL
LIN {X 0,Y 477.688,Z 564.063,A -85,B 0,C 180,E1 8660.269,E2 8660.269} C_VEL
LIN {X 0,Y 472.35,Z 553.588,A -85,B 0,C 180,E1 8657.62,E2 8657.62} C_VEL
LIN {X 0,Y 467.644,Z 544.664,A -85,B 0,C 180,E1 8654.804,E2 8654.804} C_VEL
LIN {X 0,Y 464.283,Z 538.514,A -85,B 0,C 180,E1 8652.311,E2 8652.311} C_VEL
LIN {X 0,Y 461.959,Z 534.167,A -85,B 0,C 180,E1 8650.097,E2 8650.097} C_VEL
LIN {X 0,Y 460.474,Z 531.201,A -85,B 0,C 180,E1 8648.24,E2 8648.24} C_VEL
LIN {X 0,Y 458.602,Z 527.135,A -85,B 0,C 180,E1 8644.126,E2 8644.126} C_VEL
LIN {X 0,Y 458.636,Z 526.77,A -85,B 0,C 180,E1 8640.125,E2 8640.125} C_VEL
LIN {X 0,Y 459.996,Z 528.027,A -85,B 0,C 180,E1 8637.01,E2 8637.01} C_VEL
LIN {X 0,Y 463.231,Z 532.943,A -85,B 0,C 180,E1 8633.12,E2 8633.12} C_VEL
LIN {X 0,Y 466.207,Z 537.565,A -85,B 0,C 180,E1 8630.681,E2 8630.681} C_VEL
LIN {X 0,Y 469.663,Z 543.057,A -85,B 0,C 180,E1 8628.394,E2 8628.394} C_VEL
LIN {X 0,Y 473.769,Z 549.769,A -85,B 0,C 180,E1 8626.109,E2 8626.109} C_VEL
LIN {X 0,Y 479.097,Z 559.029,A -85,B 0,C 180,E1 8623.573,E2 8623.573} C_VEL
LIN {X 0,Y 479.685,Z 560.327,A -85,B 0,C 180,E1 8623.303,E2 8623.303} C_VEL
LIN {X 0,Y 460.709,Z 780.763,A -85,B 0,C 180,E1 8619.854,E2 8619.854} C_VEL
LIN {X 0,Y 456.147,Z 831.439,A -85,B 0,C 180,E1 8619.033,E2 8619.033} C_VEL
LIN {X 0,Y 451.898,Z 859.876,A -85,B 0,C 180,E1 8618.468,E2 8618.468} C_VEL
LIN {X 0,Y 447.517,Z 881.963,A -85,B 0,C 180,E1 8617.909,E2 8617.909} C_VEL
LIN {X 0,Y 442.417,Z 903.466,A -85,B 0,C 180,E1 8617.233,E2 8617.233} C_VEL
LIN {X 0,Y 435.322,Z 929.001,A -85,B 0,C 180,E1 8616.248,E2 8616.248} C_VEL
LIN {X 0,Y 427.247,Z 953.341,A -85,B 0,C 180,E1 8615.074,E2 8615.074} C_VEL
LIN {X 0,Y 420.071,Z 972.733,A -85,B 0,C 180,E1 8613.967,E2 8613.967} C_VEL
LIN {X 0,Y 412.03,Z 992.542,A -85,B 0,C 180,E1 8612.644,E2 8612.644} C_VEL
LIN {X 0,Y 401.886,Z 1015.41,A -85,B 0,C 180,E1 8610.841,E2 8610.841} C_VEL
LIN {X 0,Y 391.471,Z 1036.559,A -85,B 0,C 180,E1 8608.83,E2 8608.83} C_VEL
LIN {X 0,Y 382.768,Z 1053.202,A -85,B 0,C 180,E1 8606.984,E2 8606.984} C_VEL
LIN {X 0,Y 373.724,Z 1069.618,A -85,B 0,C 180,E1 8604.884,E2 8604.884} C_VEL
LIN {X 0,Y 362.782,Z 1088.688,A -85,B 0,C 180,E1 8602.022,E2 8602.022} C_VEL
LIN {X 0,Y 352.56,Z 1105.568,A -85,B 0,C 180,E1 8598.971,E2 8598.971} C_VEL
LIN {X 0,Y 344.187,Z 1119.209,A -85,B 0,C 180,E1 8596.091,E2 8596.091} C_VEL
LIN {X 0,Y 336.201,Z 1132.135,A -85,B 0,C 180,E1 8592.926,E2 8592.926} C_VEL
LIN {X 0,Y 327.106,Z 1147.061,A -85,B 0,C 180,E1 8588.577,E2 8588.577} C_VEL
LIN {X 0,Y 320.443,Z 1158.34,A -85,B 0,C 180,E1 8584.603,E2 8584.603} C_VEL
LIN {X 0,Y 315.481,Z 1167.313,A -85,B 0,C 180,E1 8580.893,E2 8580.893} C_VEL
LIN {X 0,Y 311.183,Z 1175.883,A -85,B 0,C 180,E1 8576.713,E2 8576.713} C_VEL
LIN {X 0,Y 307.379,Z 1184.733,A -85,B 0,C 180,E1 8571.366,E2 8571.366} C_VEL
LIN {X 0,Y 305.51,Z 1190.237,A -85,B 0,C 180,E1 8567.122,E2 8567.122} C_VEL
LIN {X 0,Y 304.539,Z 1194.172,A -85,B 0,C 180,E1 8563.286,E2 8563.286} C_VEL
LIN {X 0,Y 304.101,Z 1197.12,A -85,B 0,C 180,E1 8559.457,E2 8559.457} C_VEL
LIN {X 0,Y 303.979,Z 1199.004,A -85,B 0,C 180,E1 8555.852,E2 8555.852} C_VEL
LIN {X 0,Y 303.974,Z 1200.007,A -85,B 0,C 180,E1 8552.262,E2 8552.262} C_VEL
LIN {X 0,Y 303.979,Z 1200.126,A -85,B 0,C 180,E1 8548.68,E2 8548.68} C_VEL
LIN {X 0,Y 303.972,Z 1199.359,A -85,B 0,C 180,E1 8545.093,E2 8545.093} C_VEL
LIN {X 0,Y 304.059,Z 1197.589,A -85,B 0,C 180,E1 8541.299,E2 8541.299} C_VEL
LIN {X 0,Y 304.416,Z 1194.833,A -85,B 0,C 180,E1 8537.48,E2 8537.48} C_VEL
LIN {X 0,Y 305.274,Z 1191.081,A -85,B 0,C 180,E1 8533.639,E2 8533.639} C_VEL
LIN {X 0,Y 306.762,Z 1186.311,A -85,B 0,C 180,E1 8529.787,E2 8529.787} C_VEL
LIN {X 0,Y 309.064,Z 1180.498,A -85,B 0,C 180,E1 8525.943,E2 8525.943} C_VEL
LIN {X 0,Y 312.427,Z 1173.239,A -85,B 0,C 180,E1 8521.936,E2 8521.936} C_VEL
LIN {X 0,Y 317.853,Z 1163.052,A -85,B 0,C 180,E1 8517.243,E2 8517.243} C_VEL
LIN {X 0,Y 324.53,Z 1151.274,A -85,B 0,C 180,E1 8512.852,E2 8512.852} C_VEL
LIN {X 0,Y 330.912,Z 1140.678,A -85,B 0,C 180,E1 8509.485,E2 8509.485} C_VEL
LIN {X 0,Y 338.21,Z 1128.798,A -85,B 0,C 180,E1 8506.227,E2 8506.227} C_VEL
LIN {X 0,Y 347.803,Z 1113.365,A -85,B 0,C 180,E1 8502.611,E2 8502.611} C_VEL
LIN {X 0,Y 358.029,Z 1096.373,A -85,B 0,C 180,E1 8499.323,E2 8499.323} C_VEL
LIN {X 0,Y 367.076,Z 1081.044,A -85,B 0,C 180,E1 8496.791,E2 8496.791} C_VEL
LIN {X 0,Y 376.402,Z 1064.671,A -85,B 0,C 180,E1 8494.46,E2 8494.46} C_VEL
LIN {X 0,Y 388.291,Z 1042.58,A -85,B 0,C 180,E1 8491.812,E2 8491.812} C_VEL
LIN {X 0,Y 397.882,Z 1023.356,A -85,B 0,C 180,E1 8489.889,E2 8489.889} C_VEL
LIN {X 0,Y 406.542,Z 1004.8,A -85,B 0,C 180,E1 8488.298,E2 8488.298} C_VEL
LIN {X 0,Y 415.824,Z 983.299,A -85,B 0,C 180,E1 8486.722,E2 8486.722} C_VEL
LIN {X 0,Y 425.06,Z 959.137,A -85,B 0,C 180,E1 8485.248,E2 8485.248} C_VEL
LIN {X 0,Y 431.969,Z 938.934,A -85,B 0,C 180,E1 8484.218,E2 8484.218} C_VEL
LIN {X 0,Y 438.264,Z 918.235,A -85,B 0,C 180,E1 8483.323,E2 8483.323} C_VEL
LIN {X 0,Y 444.488,Z 894.769,A -85,B 0,C 180,E1 8482.484,E2 8482.484} C_VEL
LIN {X 0,Y 450.397,Z 867.205,A -85,B 0,C 180,E1 8481.71,E2 8481.71} C_VEL
LIN {X 0,Y 454.194,Z 844.708,A -85,B 0,C 180,E1 8481.224,E2 8481.224} C_VEL
LIN {X 0,Y 456.989,Z 821.922,A -85,B 0,C 180,E1 8480.813,E2 8480.813} C_VEL
LIN {X 0,Y 475.518,Z 606.098,A -85,B 0,C 180,E1 8477.415,E2 8477.415} C_VEL
LIN {X 0,Y 479.538,Z 559.935,A -85,B 0,C 180,E1 8476.692,E2 8476.692} C_VEL
LIN {X 0,Y 473.825,Z 550.031,A -85,B 0,C 180,E1 8474.014,E2 8474.014} C_VEL
LIN {X 0,Y 469.671,Z 543.203,A -85,B 0,C 180,E1 8471.731,E2 8471.731} C_VEL
LIN {X 0,Y 466.852,Z 538.805,A -85,B 0,C 180,E1 8469.928,E2 8469.928} C_VEL
LIN {X 0,Y 464.801,Z 535.525,A -85,B 0,C 180,E1 8468.412,E2 8468.412} C_VEL
LIN {X 0,Y 462.458,Z 531.876,A -85,B 0,C 180,E1 8466.331,E2 8466.331} C_VEL
LIN {X 0,Y 459.533,Z 527.477,A -85,B 0,C 180,E1 8462.619,E2 8462.619} C_VEL
LIN {X 0,Y 458.116,Z 526.441,A -85,B 0,C 180,E1 8458.434,E2 8458.434} C_VEL
LIN {X 0,Y 458.507,Z 527.25,A -85,B 0,C 180,E1 8455.121,E2 8455.121} C_VEL
LIN {X 0,Y 460.809,Z 532.07,A -85,B 0,C 180,E1 8450.886,E2 8450.886} C_VEL
LIN {X 0,Y 463.142,Z 536.609,A -85,B 0,C 180,E1 8448.417,E2 8448.417} C_VEL
LIN {X 0,Y 465.527,Z 540.987,A -85,B 0,C 180,E1 8446.46,E2 8446.46} C_VEL
LIN {X 0,Y 469.008,Z 547.457,A -85,B 0,C 180,E1 8444.1,E2 8444.1} C_VEL
LIN {X 0,Y 473.305,Z 555.637,A -85,B 0,C 180,E1 8441.685,E2 8441.685} C_VEL
LIN {X 0,Y 477.578,Z 564.101,A -85,B 0,C 180,E1 8439.608,E2 8439.608} C_VEL
LIN {X 0,Y 459.122,Z 785.976,A -85,B 0,C 180,E1 8436.256,E2 8436.256} C_VEL
LIN {X 0,Y 454.854,Z 834.824,A -85,B 0,C 180,E1 8435.492,E2 8435.492} C_VEL
LIN {X 0,Y 450.839,Z 861.677,A -85,B 0,C 180,E1 8434.965,E2 8434.965} C_VEL
LIN {X 0,Y 446.472,Z 883.651,A -85,B 0,C 180,E1 8434.42,E2 8434.42} C_VEL
LIN {X 0,Y 441.09,Z 906.201,A -85,B 0,C 180,E1 8433.706,E2 8433.706} C_VEL
LIN {X 0,Y 433.393,Z 932.716,A -85,B 0,C 180,E1 8432.652,E2 8432.652} C_VEL
LIN {X 0,Y 426.921,Z 951.962,A -85,B 0,C 180,E1 8431.717,E2 8431.717} C_VEL
LIN {X 0,Y 419.849,Z 970.776,A -85,B 0,C 180,E1 8430.65,E2 8430.65} C_VEL
LIN {X 0,Y 410.912,Z 992.333,A -85,B 0,C 180,E1 8429.2,E2 8429.2} C_VEL
LIN {X 0,Y 400.375,Z 1014.941,A -85,B 0,C 180,E1 8427.355,E2 8427.355} C_VEL
LIN {X 0,Y 391.63,Z 1032.199,A -85,B 0,C 180,E1 8425.684,E2 8425.684} C_VEL
LIN {X 0,Y 382.566,Z 1048.957,A -85,B 0,C 180,E1 8423.794,E2 8423.794} C_VEL
LIN {X 0,Y 371.1,Z 1068.771,A -85,B 0,C 180,E1 8421.139,E2 8421.139} C_VEL
LIN {X 0,Y 361.327,Z 1084.603,A -85,B 0,C 180,E1 8418.584,E2 8418.584} C_VEL
LIN {X 0,Y 352.536,Z 1098.366,A -85,B 0,C 180,E1 8415.981,E2 8415.981} C_VEL
LIN {X 0,Y 342.666,Z 1113.492,A -85,B 0,C 180,E1 8412.607,E2 8412.607} C_VEL
LIN {X 0,Y 333.728,Z 1126.741,A -85,B 0,C 180,E1 8408.99,E2 8408.99} C_VEL
LIN {X 0,Y 326.669,Z 1137.34,A -85,B 0,C 180,E1 8405.561,E2 8405.561} C_VEL
LIN {X 0,Y 319.575,Z 1148.406,A -85,B 0,C 180,E1 8401.291,E2 8401.291} C_VEL
LIN {X 0,Y 313.733,Z 1157.866,A -85,B 0,C 180,E1 8396.704,E2 8396.704} C_VEL
LIN {X 0,Y 310.005,Z 1164.612,A -85,B 0,C 180,E1 8392.71,E2 8392.71} C_VEL
LIN {X 0,Y 307.088,Z 1170.76,A -85,B 0,C 180,E1 8388.215,E2 8388.215} C_VEL
LIN {X 0,Y 305.162,Z 1175.777,A -85,B 0,C 180,E1 8383.26,E2 8383.26} C_VEL
LIN {X 0,Y 304.386,Z 1178.751,A -85,B 0,C 180,E1 8379.072,E2 8379.072} C_VEL
LIN {X 0,Y 304.079,Z 1180.494,A -85,B 0,C 180,E1 8375.283,E2 8375.283} C_VEL
LIN {X 0,Y 304.005,Z 1181.303,A -85,B 0,C 180,E1 8371.697,E2 8371.697} C_VEL
LIN {X 0,Y 304.013,Z 1181.294,A -85,B 0,C 180,E1 8368.116,E2 8368.116} C_VEL
LIN {X 0,Y 304.084,Z 1180.469,A -85,B 0,C 180,E1 8364.529,E2 8364.529} C_VEL
LIN {X 0,Y 304.395,Z 1178.708,A -85,B 0,C 180,E1 8360.738,E2 8360.738} C_VEL
LIN {X 0,Y 305.196,Z 1175.714,A -85,B 0,C 180,E1 8356.55,E2 8356.55} C_VEL
LIN {X 0,Y 307.24,Z 1170.412,A -85,B 0,C 180,E1 8351.402,E2 8351.402} C_VEL
LIN {X 0,Y 310.131,Z 1164.401,A -85,B 0,C 180,E1 8347.039,E2 8347.039} C_VEL
LIN {X 0,Y 313.846,Z 1157.722,A -85,B 0,C 180,E1 8343.103,E2 8343.103} C_VEL
LIN {X 0,Y 319.729,Z 1148.207,A -85,B 0,C 180,E1 8338.517,E2 8338.517} C_VEL
LIN {X 0,Y 326.536,Z 1137.609,A -85,B 0,C 180,E1 8334.424,E2 8334.424} C_VEL
LIN {X 0,Y 333.584,Z 1127.04,A -85,B 0,C 180,E1 8330.991,E2 8330.991} C_VEL
LIN {X 0,Y 342.939,Z 1113.184,A -85,B 0,C 180,E1 8327.209,E2 8327.209} C_VEL
LIN {X 0,Y 352.582,Z 1098.421,A -85,B 0,C 180,E1 8323.92,E2 8323.92} C_VEL
LIN {X 0,Y 361.147,Z 1085.04,A -85,B 0,C 180,E1 8321.385,E2 8321.385} C_VEL
LIN {X 0,Y 370.909,Z 1069.242,A -85,B 0,C 180,E1 8318.825,E2 8318.825} C_VEL
LIN {X 0,Y 382.534,Z 1049.22,A -85,B 0,C 180,E1 8316.132,E2 8316.132} C_VEL
LIN {X 0,Y 388.916,Z 1037.652,A -85,B 0,C 180,E1 8314.785,E2 8314.785} C_VEL
LIN {X 0,Y 391.241,Z 1032.161,A -85,B 0,C 180,E1 8314.071,E2 8314.071} C_VEL
LIN {X 0,Y 395.046,Z 1018.616,A -85,B 0,C 180,E1 8311.974,E2 8311.974} C_VEL
LIN {X 0,Y 397.53,Z 1012.721,A -85,B 0,C 180,E1 8311.321,E2 8311.321} C_VEL
LIN {X 0,Y 408.025,Z 990.356,A -85,B 0,C 180,E1 8309.549,E2 8309.549} C_VEL
LIN {X 0,Y 416.481,Z 970.325,A -85,B 0,C 180,E1 8308.227,E2 8308.227} C_VEL
LIN {X 0,Y 424.068,Z 950.449,A -85,B 0,C 180,E1 8307.118,E2 8307.118} C_VEL
LIN {X 0,Y 432.189,Z 926.385,A -85,B 0,C 180,E1 8306,E2 8306} C_VEL
LIN {X 0,Y 438.743,Z 903.205,A -85,B 0,C 180,E1 8305.135,E2 8305.135} C_VEL
LIN {X 0,Y 443.754,Z 882.326,A -85,B 0,C 180,E1 8304.494,E2 8304.494} C_VEL
LIN {X 0,Y 448.368,Z 859.14,A -85,B 0,C 180,E1 8303.933,E2 8303.933} C_VEL
LIN {X 0,Y 452.406,Z 830.867,A -85,B 0,C 180,E1 8303.405,E2 8303.405} C_VEL
LIN {X 0,Y 459.979,Z 742.643,A -85,B 0,C 180,E1 8302.055,E2 8302.055} C_VEL
LIN {X 0,Y 474.821,Z 569.132,A -85,B 0,C 180,E1 8299.434,E2 8299.434} C_VEL
LIN {X 0,Y 469.363,Z 558.26,A -85,B 0,C 180,E1 8296.529,E2 8296.529} C_VEL
LIN {X 0,Y 465.432,Z 550.728,A -85,B 0,C 180,E1 8293.986,E2 8293.986} C_VEL
LIN {X 0,Y 462.8,Z 545.847,A -85,B 0,C 180,E1 8291.907,E2 8291.907} C_VEL
LIN {X 0,Y 460.75,Z 541.858,A -85,B 0,C 180,E1 8289.862,E2 8289.862} C_VEL
LIN {X 0,Y 459.326,Z 538.969,A -85,B 0,C 180,E1 8288.009,E2 8288.009} C_VEL
LIN {X 0,Y 457.598,Z 535.044,A -85,B 0,C 180,E1 8284.01,E2 8284.01} C_VEL
LIN {X 0,Y 457.659,Z 534.711,A -85,B 0,C 180,E1 8280.125,E2 8280.125} C_VEL
LIN {X 0,Y 458.938,Z 535.905,A -85,B 0,C 180,E1 8277.128,E2 8277.128} C_VEL
LIN {X 0,Y 462.038,Z 540.741,A -85,B 0,C 180,E1 8273.289,E2 8273.289} C_VEL
LIN {X 0,Y 464.876,Z 545.246,A -85,B 0,C 180,E1 8270.904,E2 8270.904} C_VEL
LIN {X 0,Y 468.254,Z 550.745,A -85,B 0,C 180,E1 8268.608,E2 8268.608} C_VEL
LIN {X 0,Y 472.339,Z 557.618,A -85,B 0,C 180,E1 8266.285,E2 8266.285} C_VEL
LIN {X 0,Y 476.709,Z 565.362,A -85,B 0,C 180,E1 8264.141,E2 8264.141} C_VEL
LIN {X 0,Y 457.615,Z 782.462,A -85,B 0,C 180,E1 8260.759,E2 8260.759} C_VEL
LIN {X 0,Y 453.033,Z 832.033,A -85,B 0,C 180,E1 8259.959,E2 8259.959} C_VEL
LIN {X 0,Y 448.721,Z 860.17,A -85,B 0,C 180,E1 8259.403,E2 8259.403} C_VEL
LIN {X 0,Y 444.298,Z 882.071,A -85,B 0,C 180,E1 8258.855,E2 8258.855} C_VEL
LIN {X 0,Y 439.127,Z 903.465,A -85,B 0,C 180,E1 8258.191,E2 8258.191} C_VEL
LIN {X 0,Y 432.087,Z 928.382,A -85,B 0,C 180,E1 8257.243,E2 8257.243} C_VEL
LIN {X 0,Y 423.846,Z 952.821,A -85,B 0,C 180,E1 8256.082,E2 8256.082} C_VEL
LIN {X 0,Y 416.552,Z 972.166,A -85,B 0,C 180,E1 8254.992,E2 8254.992} C_VEL
LIN {X 0,Y 408.433,Z 991.785,A -85,B 0,C 180,E1 8253.697,E2 8253.697} C_VEL
LIN {X 0,Y 398.587,Z 1013.584,A -85,B 0,C 180,E1 8252.007,E2 8252.007} C_VEL
LIN {X 0,Y 387.691,Z 1035.308,A -85,B 0,C 180,E1 8249.977,E2 8249.977} C_VEL
LIN {X 0,Y 378.559,Z 1052.326,A -85,B 0,C 180,E1 8248.112,E2 8248.112} C_VEL
LIN {X 0,Y 369.397,Z 1068.501,A -85,B 0,C 180,E1 8246.06,E2 8246.06} C_VEL
LIN {X 0,Y 358.2,Z 1087.47,A -85,B 0,C 180,E1 8243.238,E2 8243.238} C_VEL
LIN {X 0,Y 347.074,Z 1105.267,A -85,B 0,C 180,E1 8240.023,E2 8240.023} C_VEL
LIN {X 0,Y 338.375,Z 1118.913,A -85,B 0,C 180,E1 8237.123,E2 8237.123} C_VEL
LIN {X 0,Y 330.059,Z 1131.844,A -85,B 0,C 180,E1 8233.926,E2 8233.926} C_VEL
LIN {X 0,Y 320.529,Z 1146.782,A -85,B 0,C 180,E1 8229.521,E2 8229.521} C_VEL
LIN {X 0,Y 313.541,Z 1158.064,A -85,B 0,C 180,E1 8225.478,E2 8225.478} C_VEL
LIN {X 0,Y 308.291,Z 1167.042,A -85,B 0,C 180,E1 8221.696,E2 8221.696} C_VEL
LIN {X 0,Y 303.744,Z 1175.58,A -85,B 0,C 180,E1 8217.442,E2 8217.442} C_VEL
LIN {X 0,Y 299.659,Z 1184.488,A -85,B 0,C 180,E1 8211.933,E2 8211.933} C_VEL
LIN {X 0,Y 297.649,Z 1189.971,A -85,B 0,C 180,E1 8207.597,E2 8207.597} C_VEL
LIN {X 0,Y 296.6,Z 1193.918,A -85,B 0,C 180,E1 8203.649,E2 8203.649} C_VEL
LIN {X 0,Y 296.119,Z 1196.866,A -85,B 0,C 180,E1 8199.719,E2 8199.719} C_VEL
LIN {X 0,Y 295.983,Z 1198.756,A -85,B 0,C 180,E1 8196.011,E2 8196.011} C_VEL
LIN {X 0,Y 295.977,Z 1199.76,A -85,B 0,C 180,E1 8192.323,E2 8192.323} C_VEL
LIN {X 0,Y 295.983,Z 1199.879,A -85,B 0,C 180,E1 8188.645,E2 8188.645} C_VEL
LIN {X 0,Y 295.975,Z 1199.111,A -85,B 0,C 180,E1 8184.961,E2 8184.961} C_VEL
LIN {X 0,Y 296.072,Z 1197.337,A -85,B 0,C 180,E1 8181.063,E2 8181.063} C_VEL
LIN {X 0,Y 296.474,Z 1194.53,A -85,B 0,C 180,E1 8177.081,E2 8177.081} C_VEL
LIN {X 0,Y 297.399,Z 1190.823,A -85,B 0,C 180,E1 8173.193,E2 8173.193} C_VEL
LIN {X 0,Y 299.011,Z 1186.05,A -85,B 0,C 180,E1 8169.239,E2 8169.239} C_VEL
LIN {X 0,Y 301.469,Z 1180.233,A -85,B 0,C 180,E1 8165.297,E2 8165.297} C_VEL
LIN {X 0,Y 305.054,Z 1172.969,A -85,B 0,C 180,E1 8161.195,E2 8161.195} C_VEL
LIN {X 0,Y 310.791,Z 1162.774,A -85,B 0,C 180,E1 8156.402,E2 8156.402} C_VEL
LIN {X 0,Y 317.842,Z 1150.991,A -85,B 0,C 180,E1 8151.932,E2 8151.932} C_VEL
LIN {X 0,Y 324.898,Z 1139.798,A -85,B 0,C 180,E1 8148.337,E2 8148.337} C_VEL
LIN {X 0,Y 332.993,Z 1127.197,A -85,B 0,C 180,E1 8144.875,E2 8144.875} C_VEL
LIN {X 0,Y 344.065,Z 1109.91,A -85,B 0,C 180,E1 8140.924,E2 8140.924} C_VEL
LIN {X 0,Y 353.365,Z 1095.055,A -85,B 0,C 180,E1 8138.087,E2 8138.087} C_VEL
LIN {X 0,Y 362.736,Z 1079.672,A -85,B 0,C 180,E1 8135.565,E2 8135.565} C_VEL
LIN {X 0,Y 374.122,Z 1060.266,A -85,B 0,C 180,E1 8132.857,E2 8132.857} C_VEL
LIN {X 0,Y 384.922,Z 1040.347,A -85,B 0,C 180,E1 8130.558,E2 8130.558} C_VEL
LIN {X 0,Y 394.135,Z 1022.283,A -85,B 0,C 180,E1 8128.777,E2 8128.777} C_VEL
LIN {X 0,Y 403.38,Z 1002.855,A -85,B 0,C 180,E1 8127.136,E2 8127.136} C_VEL
LIN {X 0,Y 414.34,Z 977.445,A -85,B 0,C 180,E1 8125.346,E2 8125.346} C_VEL
LIN {X 0,Y 422.201,Z 956.98,A -85,B 0,C 180,E1 8124.149,E2 8124.149} C_VEL
LIN {X 0,Y 429.042,Z 937.196,A -85,B 0,C 180,E1 8123.164,E2 8123.164} C_VEL
LIN {X 0,Y 435.72,Z 915.423,A -85,B 0,C 180,E1 8122.25,E2 8122.25} C_VEL
LIN {X 0,Y 443.034,Z 887.092,A -85,B 0,C 180,E1 8121.296,E2 8121.296} C_VEL
LIN {X 0,Y 447.767,Z 864.426,A -85,B 0,C 180,E1 8120.702,E2 8120.702} C_VEL
LIN {X 0,Y 451.455,Z 842.377,A -85,B 0,C 180,E1 8120.241,E2 8120.241} C_VEL
LIN {X 0,Y 454.668,Z 815.021,A -85,B 0,C 180,E1 8119.762,E2 8119.762} C_VEL
LIN {X 0,Y 474.416,Z 589.118,A -85,B 0,C 180,E1 8116.235,E2 8116.235} C_VEL
LIN {X 0,Y 476.517,Z 565.195,A -85,B 0,C 180,E1 8115.851,E2 8115.851} C_VEL
LIN {X 0,Y 471.398,Z 556.061,A -85,B 0,C 180,E1 8113.305,E2 8113.305} C_VEL
LIN {X 0,Y 466.853,Z 548.442,A -85,B 0,C 180,E1 8110.614,E2 8110.614} C_VEL
LIN {X 0,Y 463.497,Z 543.212,A -85,B 0,C 180,E1 8108.186,E2 8108.186} C_VEL
LIN {X 0,Y 461.216,Z 539.608,A -85,B 0,C 180,E1 8106.098,E2 8106.098} C_VEL
LIN {X 0,Y 458.478,Z 535.376,A -85,B 0,C 180,E1 8102.5,E2 8102.5} C_VEL
LIN {X 0,Y 457.147,Z 534.382,A -85,B 0,C 180,E1 8098.496,E2 8098.496} C_VEL
LIN {X 0,Y 457.526,Z 535.274,A -85,B 0,C 180,E1 8095.111,E2 8095.111} C_VEL
LIN {X 0,Y 459.685,Z 539.88,A -85,B 0,C 180,E1 8091.053,E2 8091.053} C_VEL
LIN {X 0,Y 461.894,Z 544.307,A -85,B 0,C 180,E1 8088.639,E2 8088.639} C_VEL
LIN {X 0,Y 464.223,Z 548.698,A -85,B 0,C 180,E1 8086.675,E2 8086.675} C_VEL
LIN {X 0,Y 467.535,Z 555.028,A -85,B 0,C 180,E1 8084.367,E2 8084.367} C_VEL
LIN {X 0,Y 471.683,Z 563.125,A -85,B 0,C 180,E1 8081.971,E2 8081.971} C_VEL
LIN {X 0,Y 474.654,Z 569.348,A -85,B 0,C 180,E1 8080.45,E2 8080.45} C_VEL
LIN {X 0,Y 455.779,Z 791.073,A -85,B 0,C 180,E1 8077.115,E2 8077.115} C_VEL
LIN {X 0,Y 451.659,Z 836.425,A -85,B 0,C 180,E1 8076.405,E2 8076.405} C_VEL
LIN {X 0,Y 447.553,Z 862.662,A -85,B 0,C 180,E1 8075.888,E2 8075.888} C_VEL
LIN {X 0,Y 443.148,Z 884.296,A -85,B 0,C 180,E1 8075.354,E2 8075.354} C_VEL
LIN {X 0,Y 437.242,Z 908.414,A -85,B 0,C 180,E1 8074.593,E2 8074.593} C_VEL
LIN {X 0,Y 429.777,Z 933.289,A -85,B 0,C 180,E1 8073.599,E2 8073.599} C_VEL
LIN {X 0,Y 423.177,Z 952.476,A -85,B 0,C 180,E1 8072.674,E2 8072.674} C_VEL
LIN {X 0,Y 415.964,Z 971.244,A -85,B 0,C 180,E1 8071.616,E2 8071.616} C_VEL
LIN {X 0,Y 406.838,Z 992.766,A -85,B 0,C 180,E1 8070.177,E2 8070.177} C_VEL
LIN {X 0,Y 396.285,Z 1014.876,A -85,B 0,C 180,E1 8068.382,E2 8068.382} C_VEL
LIN {X 0,Y 387.106,Z 1032.553,A -85,B 0,C 180,E1 8066.677,E2 8066.677} C_VEL
LIN {X 0,Y 377.972,Z 1048.998,A -85,B 0,C 180,E1 8064.828,E2 8064.828} C_VEL
LIN {X 0,Y 366.603,Z 1068.173,A -85,B 0,C 180,E1 8062.275,E2 8062.275} C_VEL
LIN {X 0,Y 355.949,Z 1084.905,A -85,B 0,C 180,E1 8059.575,E2 8059.575} C_VEL
LIN {X 0,Y 347.095,Z 1098.313,A -85,B 0,C 180,E1 8057.029,E2 8057.029} C_VEL
LIN {X 0,Y 336.599,Z 1113.823,A -85,B 0,C 180,E1 8053.546,E2 8053.546} C_VEL
LIN {X 0,Y 327.342,Z 1127.017,A -85,B 0,C 180,E1 8049.901,E2 8049.901} C_VEL
LIN {X 0,Y 319.981,Z 1137.61,A -85,B 0,C 180,E1 8046.421,E2 8046.421} C_VEL
LIN {X 0,Y 312.407,Z 1148.885,A -85,B 0,C 180,E1 8041.987,E2 8041.987} C_VEL
LIN {X 0,Y 306.389,Z 1158.129,A -85,B 0,C 180,E1 8037.397,E2 8037.397} C_VEL
LIN {X 0,Y 302.485,Z 1164.783,A -85,B 0,C 180,E1 8033.37,E2 8033.37} C_VEL
LIN {X 0,Y 299.331,Z 1171.017,A -85,B 0,C 180,E1 8028.704,E2 8028.704} C_VEL
LIN {X 0,Y 297.251,Z 1176.077,A -85,B 0,C 180,E1 8023.556,E2 8023.556} C_VEL
LIN {X 0,Y 296.42,Z 1179.002,A -85,B 0,C 180,E1 8019.318,E2 8019.318} C_VEL
LIN {X 0,Y 296.09,Z 1180.743,A -85,B 0,C 180,E1 8015.426,E2 8015.426} C_VEL
LIN {X 0,Y 296.01,Z 1181.55,A -85,B 0,C 180,E1 8011.743,E2 8011.743} C_VEL
LIN {X 0,Y 296.016,Z 1181.563,A -85,B 0,C 180,E1 8008.258,E2 8008.258} C_VEL
LIN {X 0,Y 296.086,Z 1180.781,A -85,B 0,C 180,E1 8004.575,E2 8004.575} C_VEL
LIN {X 0,Y 296.387,Z 1179.173,A -85,B 0,C 180,E1 8000.877,E2 8000.877} C_VEL
LIN {X 0,Y 297.134,Z 1176.421,A -85,B 0,C 180,E1 7996.773,E2 7996.773} C_VEL
LIN {X 0,Y 298.788,Z 1172.228,A -85,B 0,C 180,E1 7992.271,E2 7992.271} C_VEL
LIN {X 0,Y 302.106,Z 1165.532,A -85,B 0,C 180,E1 7987.012,E2 7987.012} C_VEL
LIN {X 0,Y 306.088,Z 1158.661,A -85,B 0,C 180,E1 7982.786,E2 7982.786} C_VEL
LIN {X 0,Y 311.335,Z 1150.48,A -85,B 0,C 180,E1 7978.65,E2 7978.65} C_VEL
LIN {X 0,Y 319.167,Z 1138.877,A -85,B 0,C 180,E1 7973.917,E2 7973.917} C_VEL
LIN {X 0,Y 326.417,Z 1128.427,A -85,B 0,C 180,E1 7970.421,E2 7970.421} C_VEL
LIN {X 0,Y 334.255,Z 1117.197,A -85,B 0,C 180,E1 7967.232,E2 7967.232} C_VEL
LIN {X 0,Y 344.544,Z 1102.335,A -85,B 0,C 180,E1 7963.685,E2 7963.685} C_VEL
LIN {X 0,Y 355.081,Z 1086.39,A -85,B 0,C 180,E1 7960.578,E2 7960.578} C_VEL
LIN {X 0,Y 364.093,Z 1072.272,A -85,B 0,C 180,E1 7958.241,E2 7958.241} C_VEL
LIN {X 0,Y 374.99,Z 1054.423,A -85,B 0,C 180,E1 7955.729,E2 7955.729} C_VEL
LIN {X 0,Y 385.945,Z 1034.955,A -85,B 0,C 180,E1 7953.467,E2 7953.467} C_VEL
LIN {X 0,Y 395.084,Z 1017.513,A -85,B 0,C 180,E1 7951.751,E2 7951.751} C_VEL
LIN {X 0,Y 397.53,Z 1012.721,A -85,B 0,C 180,E1 7951.321,E2 7951.321} C_VEL
LIN {X 0,Y 399.992,Z 1006.826,A -85,B 0,C 180,E1 7950.687,E2 7950.687} C_VEL
LIN {X 0,Y 403.95,Z 992.251,A -85,B 0,C 180,E1 7948.793,E2 7948.793} C_VEL
LIN {X 0,Y 406.225,Z 986.024,A -85,B 0,C 180,E1 7948.227,E2 7948.227} C_VEL
LIN {X 0,Y 414.569,Z 966.331,A -85,B 0,C 180,E1 7946.979,E2 7946.979} C_VEL
LIN {X 0,Y 424.199,Z 940.519,A -85,B 0,C 180,E1 7945.633,E2 7945.633} C_VEL
LIN {X 0,Y 430.994,Z 919.378,A -85,B 0,C 180,E1 7944.736,E2 7944.736} C_VEL
LIN {X 0,Y 436.761,Z 898.79,A -85,B 0,C 180,E1 7944.017,E2 7944.017} C_VEL
LIN {X 0,Y 442.473,Z 874.637,A -85,B 0,C 180,E1 7943.332,E2 7943.332} C_VEL
LIN {X 0,Y 447.157,Z 848.408,A -85,B 0,C 180,E1 7942.766,E2 7942.766} C_VEL
LIN {X 0,Y 450.008,Z 826.195,A -85,B 0,C 180,E1 7942.378,E2 7942.378} C_VEL
LIN {X 0,Y 469.952,Z 597.833,A -85,B 0,C 180,E1 7938.947,E2 7938.947} C_VEL
LIN {X 0,Y 472.024,Z 574.465,A -85,B 0,C 180,E1 7938.591,E2 7938.591} C_VEL
LIN {X 0,Y 467.453,Z 565.085,A -85,B 0,C 180,E1 7936.018,E2 7936.018} C_VEL
LIN {X 0,Y 463.945,Z 558.142,A -85,B 0,C 180,E1 7933.65,E2 7933.65} C_VEL
LIN {X 0,Y 461.475,Z 553.422,A -85,B 0,C 180,E1 7931.625,E2 7931.625} C_VEL
LIN {X 0,Y 459.565,Z 549.578,A -85,B 0,C 180,E1 7929.644,E2 7929.644} C_VEL
LIN {X 0,Y 458.236,Z 546.804,A -85,B 0,C 180,E1 7927.85,E2 7927.85} C_VEL
LIN {X 0,Y 456.624,Z 542.992,A -85,B 0,C 180,E1 7924.018,E2 7924.018} C_VEL
LIN {X 0,Y 456.679,Z 542.652,A -85,B 0,C 180,E1 7920.125,E2 7920.125} C_VEL
LIN {X 0,Y 457.882,Z 543.783,A -85,B 0,C 180,E1 7917.246,E2 7917.246} C_VEL
LIN {X 0,Y 460.909,Z 548.658,A -85,B 0,C 180,E1 7913.398,E2 7913.398} C_VEL
LIN {X 0,Y 463.628,Z 553.074,A -85,B 0,C 180,E1 7911.067,E2 7911.067} C_VEL
LIN {X 0,Y 467.045,Z 558.744,A -85,B 0,C 180,E1 7908.703,E2 7908.703} C_VEL
LIN {X 0,Y 471.764,Z 566.911,A -85,B 0,C 180,E1 7906.018,E2 7906.018} C_VEL
LIN {X 0,Y 473.802,Z 570.875,A -85,B 0,C 180,E1 7904.979,E2 7904.979} C_VEL
LIN {X 0,Y 453.763,Z 794.074,A -85,B 0,C 180,E1 7901.522,E2 7901.522} C_VEL
LIN {X 0,Y 449.708,Z 835.443,A -85,B 0,C 180,E1 7900.849,E2 7900.849} C_VEL
LIN {X 0,Y 445.421,Z 861.755,A -85,B 0,C 180,E1 7900.323,E2 7900.323} C_VEL
LIN {X 0,Y 441.003,Z 883.054,A -85,B 0,C 180,E1 7899.79,E2 7899.79} C_VEL
LIN {X 0,Y 435.574,Z 904.96,A -85,B 0,C 180,E1 7899.112,E2 7899.112} C_VEL
LIN {X 0,Y 427.436,Z 932.424,A -85,B 0,C 180,E1 7898.049,E2 7898.049} C_VEL
LIN {X 0,Y 419.927,Z 954.061,A -85,B 0,C 180,E1 7897.014,E2 7897.014} C_VEL
LIN {X 0,Y 412.356,Z 973.608,A -85,B 0,C 180,E1 7895.913,E2 7895.913} C_VEL
LIN {X 0,Y 403.613,Z 994.138,A -85,B 0,C 180,E1 7894.552,E2 7894.552} C_VEL
LIN {X 0,Y 391.955,Z 1018.72,A -85,B 0,C 180,E1 7892.591,E2 7892.591} C_VEL
LIN {X 0,Y 382.433,Z 1037.073,A -85,B 0,C 180,E1 7890.837,E2 7890.837} C_VEL
LIN {X 0,Y 373.259,Z 1053.641,A -85,B 0,C 180,E1 7889.004,E2 7889.004} C_VEL
LIN {X 0,Y 363.137,Z 1070.955,A -85,B 0,C 180,E1 7886.774,E2 7886.774} C_VEL
LIN {X 0,Y 350.434,Z 1091.461,A -85,B 0,C 180,E1 7883.595,E2 7883.595} C_VEL
LIN {X 0,Y 340.664,Z 1106.545,A -85,B 0,C 180,E1 7880.792,E2 7880.792} C_VEL
LIN {X 0,Y 331.722,Z 1120.058,A -85,B 0,C 180,E1 7877.858,E2 7877.858} C_VEL
LIN {X 0,Y 321.473,Z 1135.435,A -85,B 0,C 180,E1 7873.915,E2 7873.915} C_VEL
LIN {X 0,Y 312.615,Z 1148.633,A -85,B 0,C 180,E1 7869.768,E2 7869.768} C_VEL
LIN {X 0,Y 306.103,Z 1158.742,A -85,B 0,C 180,E1 7866.012,E2 7866.012} C_VEL
LIN {X 0,Y 300.19,Z 1168.453,A -85,B 0,C 180,E1 7861.753,E2 7861.753} C_VEL
LIN {X 0,Y 294.551,Z 1178.732,A -85,B 0,C 180,E1 7856.186,E2 7856.186} C_VEL
LIN {X 0,Y 291.509,Z 1185.279,A -85,B 0,C 180,E1 7851.742,E2 7851.742} C_VEL
LIN {X 0,Y 289.664,Z 1190.149,A -85,B 0,C 180,E1 7847.683,E2 7847.683} C_VEL
LIN {X 0,Y 288.63,Z 1193.833,A -85,B 0,C 180,E1 7843.829,E2 7843.829} C_VEL
LIN {X 0,Y 288.124,Z 1196.736,A -85,B 0,C 180,E1 7839.79,E2 7839.79} C_VEL
LIN {X 0,Y 287.988,Z 1198.507,A -85,B 0,C 180,E1 7836.178,E2 7836.178} C_VEL
LIN {X 0,Y 287.981,Z 1199.488,A -85,B 0,C 180,E1 7832.587,E2 7832.587} C_VEL
LIN {X 0,Y 287.985,Z 1199.655,A -85,B 0,C 180,E1 7828.806,E2 7828.806} C_VEL
LIN {X 0,Y 287.978,Z 1198.862,A -85,B 0,C 180,E1 7824.82,E2 7824.82} C_VEL
LIN {X 0,Y 288.085,Z 1197.086,A -85,B 0,C 180,E1 7820.813,E2 7820.813} C_VEL
LIN {X 0,Y 288.519,Z 1194.324,A -85,B 0,C 180,E1 7816.777,E2 7816.777} C_VEL
LIN {X 0,Y 289.532,Z 1190.565,A -85,B 0,C 180,E1 7812.722,E2 7812.722} C_VEL
LIN {X 0,Y 291.284,Z 1185.789,A -85,B 0,C 180,E1 7808.662,E2 7808.662} C_VEL
LIN {X 0,Y 293.904,Z 1179.967,A -85,B 0,C 180,E1 7804.617,E2 7804.617} C_VEL
LIN {X 0,Y 297.728,Z 1172.701,A -85,B 0,C 180,E1 7800.417,E2 7800.417} C_VEL
LIN {X 0,Y 303.795,Z 1162.496,A -85,B 0,C 180,E1 7795.521,E2 7795.521} C_VEL
LIN {X 0,Y 311.233,Z 1150.709,A -85,B 0,C 180,E1 7790.973,E2 7790.973} C_VEL
LIN {X 0,Y 318.616,Z 1139.511,A -85,B 0,C 180,E1 7787.324,E2 7787.324} C_VEL
LIN {X 0,Y 327.658,Z 1126.06,A -85,B 0,C 180,E1 7783.604,E2 7783.604} C_VEL
LIN {X 0,Y 338.595,Z 1109.603,A -85,B 0,C 180,E1 7779.844,E2 7779.844} C_VEL
LIN {X 0,Y 348.145,Z 1094.876,A -85,B 0,C 180,E1 7777.02,E2 7777.02} C_VEL
LIN {X 0,Y 357.322,Z 1080.291,A -85,B 0,C 180,E1 7774.615,E2 7774.615} C_VEL
LIN {X 0,Y 367.866,Z 1062.848,A -85,B 0,C 180,E1 7772.148,E2 7772.148} C_VEL
LIN {X 0,Y 380.084,Z 1041.217,A -85,B 0,C 180,E1 7769.606,E2 7769.606} C_VEL
LIN {X 0,Y 389.854,Z 1022.572,A -85,B 0,C 180,E1 7767.768,E2 7767.768} C_VEL
LIN {X 0,Y 398.937,Z 1003.966,A -85,B 0,C 180,E1 7766.197,E2 7766.197} C_VEL
LIN {X 0,Y 409.432,Z 980.568,A -85,B 0,C 180,E1 7764.53,E2 7764.53} C_VEL
LIN {X 0,Y 418.303,Z 958.069,A -85,B 0,C 180,E1 7763.208,E2 7763.208} C_VEL
LIN {X 0,Y 425.499,Z 937.749,A -85,B 0,C 180,E1 7762.201,E2 7762.201} C_VEL
LIN {X 0,Y 432.084,Z 916.772,A -85,B 0,C 180,E1 7761.324,E2 7761.324} C_VEL
LIN {X 0,Y 439.245,Z 890.195,A -85,B 0,C 180,E1 7760.422,E2 7760.422} C_VEL
LIN {X 0,Y 444.556,Z 865.441,A -85,B 0,C 180,E1 7759.769,E2 7759.769} C_VEL
LIN {X 0,Y 448.332,Z 843.458,A -85,B 0,C 180,E1 7759.312,E2 7759.312} C_VEL
LIN {X 0,Y 451.366,Z 818.853,A -85,B 0,C 180,E1 7758.879,E2 7758.879} C_VEL
LIN {X 0,Y 471.265,Z 596.646,A -85,B 0,C 180,E1 7755.425,E2 7755.425} C_VEL
LIN {X 0,Y 473.641,Z 570.509,A -85,B 0,C 180,E1 7755.019,E2 7755.019} C_VEL
LIN {X 0,Y 468.757,Z 561.838,A -85,B 0,C 180,E1 7752.441,E2 7752.441} C_VEL
LIN {X 0,Y 464.931,Z 555.365,A -85,B 0,C 180,E1 7750.032,E2 7750.032} C_VEL
LIN {X 0,Y 462.2,Z 550.899,A -85,B 0,C 180,E1 7747.958,E2 7747.958} C_VEL
LIN {X 0,Y 459.981,Z 547.34,A -85,B 0,C 180,E1 7745.864,E2 7745.864} C_VEL
LIN {X 0,Y 457.425,Z 543.275,A -85,B 0,C 180,E1 7742.38,E2 7742.38} C_VEL
LIN {X 0,Y 456.162,Z 542.323,A -85,B 0,C 180,E1 7738.367,E2 7738.367} C_VEL
LIN {X 0,Y 456.514,Z 543.158,A -85,B 0,C 180,E1 7735.226,E2 7735.226} C_VEL
LIN {X 0,Y 458.566,Z 547.69,A -85,B 0,C 180,E1 7731.22,E2 7731.22} C_VEL
LIN {X 0,Y 460.709,Z 552.12,A -85,B 0,C 180,E1 7728.807,E2 7728.807} C_VEL
LIN {X 0,Y 462.92,Z 556.408,A -85,B 0,C 180,E1 7726.891,E2 7726.891} C_VEL
LIN {X 0,Y 466.073,Z 562.599,A -85,B 0,C 180,E1 7724.636,E2 7724.636} C_VEL
LIN {X 0,Y 470.179,Z 570.827,A -85,B 0,C 180,E1 7722.2,E2 7722.2} C_VEL
LIN {X 0,Y 471.836,Z 574.631,A -85,B 0,C 180,E1 7721.301,E2 7721.301} C_VEL
LIN {X 0,Y 452.439,Z 797.368,A -85,B 0,C 180,E1 7717.968,E2 7717.968} C_VEL
LIN {X 0,Y 448.59,Z 837.575,A -85,B 0,C 180,E1 7717.336,E2 7717.336} C_VEL
LIN {X 0,Y 444.502,Z 863.015,A -85,B 0,C 180,E1 7716.838,E2 7716.838} C_VEL
LIN {X 0,Y 439.999,Z 884.695,A -85,B 0,C 180,E1 7716.309,E2 7716.309} C_VEL
LIN {X 0,Y 433.883,Z 909.159,A -85,B 0,C 180,E1 7715.543,E2 7715.543} C_VEL
LIN {X 0,Y 426.281,Z 933.862,A -85,B 0,C 180,E1 7714.562,E2 7714.562} C_VEL
LIN {X 0,Y 419.554,Z 952.99,A -85,B 0,C 180,E1 7713.648,E2 7713.648} C_VEL
LIN {X 0,Y 411.838,Z 972.601,A -85,B 0,C 180,E1 7712.546,E2 7712.546} C_VEL
LIN {X 0,Y 401.824,Z 995.486,A -85,B 0,C 180,E1 7711.004,E2 7711.004} C_VEL
LIN {X 0,Y 391.443,Z 1016.508,A -85,B 0,C 180,E1 7709.278,E2 7709.278} C_VEL
LIN {X 0,Y 382.371,Z 1033.507,A -85,B 0,C 180,E1 7707.632,E2 7707.632} C_VEL
LIN {X 0,Y 371.76,Z 1052.065,A -85,B 0,C 180,E1 7705.524,E2 7705.524} C_VEL
LIN {X 0,Y 359.857,Z 1071.207,A -85,B 0,C 180,E1 7702.887,E2 7702.887} C_VEL
LIN {X 0,Y 350.065,Z 1086.12,A -85,B 0,C 180,E1 7700.435,E2 7700.435} C_VEL
LIN {X 0,Y 340.504,Z 1100.115,A -85,B 0,C 180,E1 7697.731,E2 7697.731} C_VEL
LIN {X 0,Y 328.846,Z 1116.53,A -85,B 0,C 180,E1 7693.888,E2 7693.888} C_VEL
LIN {X 0,Y 320.227,Z 1128.407,A -85,B 0,C 180,E1 7690.501,E2 7690.501} C_VEL
LIN {X 0,Y 312.305,Z 1139.383,A -85,B 0,C 180,E1 7686.777,E2 7686.777} C_VEL
LIN {X 0,Y 304.134,Z 1150.918,A -85,B 0,C 180,E1 7681.959,E2 7681.959} C_VEL
LIN {X 0,Y 298.867,Z 1158.73,A -85,B 0,C 180,E1 7677.93,E2 7677.93} C_VEL
LIN {X 0,Y 294.787,Z 1165.334,A -85,B 0,C 180,E1 7673.806,E2 7673.806} C_VEL
LIN {X 0,Y 291.272,Z 1171.976,A -85,B 0,C 180,E1 7668.618,E2 7668.618} C_VEL
LIN {X 0,Y 289.262,Z 1176.584,A -85,B 0,C 180,E1 7663.595,E2 7663.595} C_VEL
LIN {X 0,Y 288.433,Z 1179.359,A -85,B 0,C 180,E1 7659.377,E2 7659.377} C_VEL
LIN {X 0,Y 288.093,Z 1181.055,A -85,B 0,C 180,E1 7655.377,E2 7655.377} C_VEL
LIN {X 0,Y 288.013,Z 1181.819,A -85,B 0,C 180,E1 7651.592,E2 7651.592} C_VEL
LIN {X 0,Y 288.022,Z 1181.767,A -85,B 0,C 180,E1 7647.812,E2 7647.812} C_VEL
LIN {X 0,Y 288.129,Z 1180.836,A -85,B 0,C 180,E1 7643.825,E2 7643.825} C_VEL
LIN {X 0,Y 288.591,Z 1178.777,A -85,B 0,C 180,E1 7639.419,E2 7639.419} C_VEL
LIN {X 0,Y 290.041,Z 1174.651,A -85,B 0,C 180,E1 7633.991,E2 7633.991} C_VEL
LIN {X 0,Y 292.249,Z 1169.947,A -85,B 0,C 180,E1 7629.576,E2 7629.576} C_VEL
LIN {X 0,Y 295.401,Z 1164.332,A -85,B 0,C 180,E1 7625.397,E2 7625.397} C_VEL
LIN {X 0,Y 300.646,Z 1156.195,A -85,B 0,C 180,E1 7620.514,E2 7620.514} C_VEL
LIN {X 0,Y 307.555,Z 1146.069,A -85,B 0,C 180,E1 7615.776,E2 7615.776} C_VEL
LIN {X 0,Y 314.463,Z 1136.44,A -85,B 0,C 180,E1 7612.051,E2 7612.051} C_VEL
LIN {X 0,Y 323.841,Z 1123.661,A -85,B 0,C 180,E1 7607.934,E2 7607.934} C_VEL
LIN {X 0,Y 334.09,Z 1109.312,A -85,B 0,C 180,E1 7604.214,E2 7604.214} C_VEL
LIN {X 0,Y 343.11,Z 1096.478,A -85,B 0,C 180,E1 7601.416,E2 7601.416} C_VEL
LIN {X 0,Y 353.887,Z 1080.657,A -85,B 0,C 180,E1 7598.498,E2 7598.498} C_VEL
LIN {X 0,Y 365.671,Z 1062.16,A -85,B 0,C 180,E1 7595.699,E2 7595.699} C_VEL
LIN {X 0,Y 375.048,Z 1046.604,A -85,B 0,C 180,E1 7593.717,E2 7593.717} C_VEL
LIN {X 0,Y 384.504,Z 1029.907,A -85,B 0,C 180,E1 7591.893,E2 7591.893} C_VEL
LIN {X 0,Y 395.706,Z 1008.522,A -85,B 0,C 180,E1 7589.924,E2 7589.924} C_VEL
LIN {X 0,Y 405.161,Z 988.404,A -85,B 0,C 180,E1 7588.39,E2 7588.39} C_VEL
LIN {X 0,Y 406.225,Z 986.024,A -85,B 0,C 180,E1 7588.227,E2 7588.227} C_VEL
LIN {X 0,Y 408.665,Z 979.732,A -85,B 0,C 180,E1 7587.684,E2 7587.684} C_VEL
LIN {X 0,Y 412.505,Z 964.29,A -85,B 0,C 180,E1 7585.965,E2 7585.965} C_VEL
LIN {X 0,Y 414.63,Z 957.714,A -85,B 0,C 180,E1 7585.48,E2 7585.48} C_VEL
LIN {X 0,Y 421.959,Z 937.678,A -85,B 0,C 180,E1 7584.5,E2 7584.5} C_VEL
LIN {X 0,Y 428.532,Z 917.31,A -85,B 0,C 180,E1 7583.661,E2 7583.661} C_VEL
LIN {X 0,Y 435.415,Z 892.64,A -85,B 0,C 180,E1 7582.836,E2 7582.836} C_VEL
LIN {X 0,Y 441.131,Z 866.639,A -85,B 0,C 180,E1 7582.173,E2 7582.173} C_VEL
LIN {X 0,Y 444.859,Z 845.01,A -85,B 0,C 180,E1 7581.737,E2 7581.737} C_VEL
LIN {X 0,Y 447.867,Z 820.519,A -85,B 0,C 180,E1 7581.324,E2 7581.324} C_VEL
LIN {X 0,Y 468.197,Z 592.155,A -85,B 0,C 180,E1 7577.921,E2 7577.921} C_VEL
LIN {X 0,Y 469.281,Z 579.603,A -85,B 0,C 180,E1 7577.707,E2 7577.707} C_VEL
LIN {X 0,Y 465.212,Z 571.169,A -85,B 0,C 180,E1 7575.266,E2 7575.266} C_VEL
LIN {X 0,Y 462.314,Z 565.26,A -85,B 0,C 180,E1 7573.19,E2 7573.19} C_VEL
LIN {X 0,Y 460.097,Z 560.871,A -85,B 0,C 180,E1 7571.279,E2 7571.279} C_VEL
LIN {X 0,Y 458.329,Z 557.18,A -85,B 0,C 180,E1 7569.354,E2 7569.354} C_VEL
LIN {X 0,Y 457.217,Z 554.735,A -85,B 0,C 180,E1 7567.793,E2 7567.793} C_VEL
LIN {X 0,Y 455.622,Z 550.902,A -85,B 0,C 180,E1 7563.901,E2 7563.901} C_VEL
LIN {X 0,Y 455.729,Z 550.619,A -85,B 0,C 180,E1 7560,E2 7560} C_VEL
LIN {X 0,Y 456.828,Z 551.66,A -85,B 0,C 180,E1 7557.366,E2 7557.366} C_VEL
LIN {X 0,Y 459.727,Z 556.456,A -85,B 0,C 180,E1 7553.569,E2 7553.569} C_VEL
LIN {X 0,Y 462.307,Z 560.754,A -85,B 0,C 180,E1 7551.292,E2 7551.292} C_VEL
LIN {X 0,Y 465.648,Z 566.429,A -85,B 0,C 180,E1 7548.92,E2 7548.92} C_VEL
LIN {X 0,Y 470.282,Z 574.637,A -85,B 0,C 180,E1 7546.224,E2 7546.224} C_VEL
LIN {X 0,Y 471.002,Z 576.239,A -85,B 0,C 180,E1 7545.83,E2 7545.83} C_VEL
LIN {X 0,Y 450.366,Z 801.51,A -85,B 0,C 180,E1 7542.362,E2 7542.362} C_VEL
LIN {X 0,Y 446.552,Z 837.7,A -85,B 0,C 180,E1 7541.768,E2 7541.768} C_VEL
LIN {X 0,Y 442.463,Z 862.175,A -85,B 0,C 180,E1 7541.281,E2 7541.281} C_VEL
LIN {X 0,Y 437.953,Z 883.493,A -85,B 0,C 180,E1 7540.754,E2 7540.754} C_VEL
LIN {X 0,Y 432.135,Z 906.457,A -85,B 0,C 180,E1 7540.048,E2 7540.048} C_VEL
LIN {X 0,Y 424.049,Z 932.992,A -85,B 0,C 180,E1 7539.025,E2 7539.025} C_VEL
LIN {X 0,Y 416.68,Z 953.82,A -85,B 0,C 180,E1 7538.041,E2 7538.041} C_VEL
LIN {X 0,Y 409.172,Z 972.866,A -85,B 0,C 180,E1 7536.984,E2 7536.984} C_VEL
LIN {X 0,Y 400.978,Z 991.804,A -85,B 0,C 180,E1 7535.753,E2 7535.753} C_VEL
LIN {X 0,Y 390.198,Z 1014.555,A -85,B 0,C 180,E1 7534.011,E2 7534.011} C_VEL
LIN {X 0,Y 379.122,Z 1035.475,A -85,B 0,C 180,E1 7532.068,E2 7532.068} C_VEL
LIN {X 0,Y 369.438,Z 1052.561,A -85,B 0,C 180,E1 7530.207,E2 7530.207} C_VEL
LIN {X 0,Y 359.343,Z 1069.39,A -85,B 0,C 180,E1 7528.066,E2 7528.066} C_VEL
LIN {X 0,Y 347.192,Z 1088.628,A -85,B 0,C 180,E1 7525.161,E2 7525.161} C_VEL
LIN {X 0,Y 335.917,Z 1105.455,A -85,B 0,C 180,E1 7522.072,E2 7522.072} C_VEL
LIN {X 0,Y 326.592,Z 1119.044,A -85,B 0,C 180,E1 7519.13,E2 7519.13} C_VEL
LIN {X 0,Y 317.191,Z 1132.574,A -85,B 0,C 180,E1 7515.689,E2 7515.689} C_VEL
LIN {X 0,Y 306.902,Z 1147.291,A -85,B 0,C 180,E1 7511.155,E2 7511.155} C_VEL
LIN {X 0,Y 299.631,Z 1157.993,A -85,B 0,C 180,E1 7507.157,E2 7507.157} C_VEL
LIN {X 0,Y 293.58,Z 1167.343,A -85,B 0,C 180,E1 7503.019,E2 7503.019} C_VEL
LIN {X 0,Y 288.003,Z 1176.877,A -85,B 0,C 180,E1 7497.949,E2 7497.949} C_VEL
LIN {X 0,Y 284.036,Z 1184.547,A -85,B 0,C 180,E1 7492.732,E2 7492.732} C_VEL
LIN {X 0,Y 281.901,Z 1189.675,A -85,B 0,C 180,E1 7488.401,E2 7488.401} C_VEL
LIN {X 0,Y 280.706,Z 1193.579,A -85,B 0,C 180,E1 7484.227,E2 7484.227} C_VEL
LIN {X 0,Y 280.145,Z 1196.485,A -85,B 0,C 180,E1 7480.072,E2 7480.072} C_VEL
LIN {X 0,Y 279.993,Z 1198.259,A -85,B 0,C 180,E1 7476.355,E2 7476.355} C_VEL
LIN {X 0,Y 279.984,Z 1199.241,A -85,B 0,C 180,E1 7472.661,E2 7472.661} C_VEL
LIN {X 0,Y 279.99,Z 1199.408,A -85,B 0,C 180,E1 7468.772,E2 7468.772} C_VEL
LIN {X 0,Y 279.982,Z 1198.614,A -85,B 0,C 180,E1 7464.672,E2 7464.672} C_VEL
LIN {X 0,Y 280.101,Z 1196.835,A -85,B 0,C 180,E1 7460.548,E2 7460.548} C_VEL
LIN {X 0,Y 280.58,Z 1194.069,A -85,B 0,C 180,E1 7456.396,E2 7456.396} C_VEL
LIN {X 0,Y 281.677,Z 1190.307,A -85,B 0,C 180,E1 7452.225,E2 7452.225} C_VEL
LIN {X 0,Y 283.604,Z 1185.473,A -85,B 0,C 180,E1 7448.011,E2 7448.011} C_VEL
LIN {X 0,Y 286.555,Z 1179.386,A -85,B 0,C 180,E1 7443.695,E2 7443.695} C_VEL
LIN {X 0,Y 291.143,Z 1171.328,A -85,B 0,C 180,E1 7438.992,E2 7438.992} C_VEL
LIN {X 0,Y 298.075,Z 1160.319,A -85,B 0,C 180,E1 7433.815,E2 7433.815} C_VEL
LIN {X 0,Y 305.058,Z 1149.896,A -85,B 0,C 180,E1 7429.781,E2 7429.781} C_VEL
LIN {X 0,Y 312.854,Z 1138.633,A -85,B 0,C 180,E1 7426.089,E2 7426.089} C_VEL
LIN {X 0,Y 323.188,Z 1123.987,A -85,B 0,C 180,E1 7422.054,E2 7422.054} C_VEL
LIN {X 0,Y 334.307,Z 1107.717,A -85,B 0,C 180,E1 7418.407,E2 7418.407} C_VEL
LIN {X 0,Y 343.709,Z 1093.696,A -85,B 0,C 180,E1 7415.744,E2 7415.744} C_VEL
LIN {X 0,Y 353.772,Z 1078.176,A -85,B 0,C 180,E1 7413.217,E2 7413.217} C_VEL
LIN {X 0,Y 366.721,Z 1057.085,A -85,B 0,C 180,E1 7410.35,E2 7410.35} C_VEL
LIN {X 0,Y 377.055,Z 1038.989,A -85,B 0,C 180,E1 7408.309,E2 7408.309} C_VEL
LIN {X 0,Y 386.407,Z 1021.503,A -85,B 0,C 180,E1 7406.616,E2 7406.616} C_VEL
LIN {X 0,Y 396.442,Z 1001.312,A -85,B 0,C 180,E1 7404.945,E2 7404.945} C_VEL
LIN {X 0,Y 407.54,Z 976.474,A -85,B 0,C 180,E1 7403.246,E2 7403.246} C_VEL
LIN {X 0,Y 415.513,Z 956.521,A -85,B 0,C 180,E1 7402.111,E2 7402.111} C_VEL
LIN {X 0,Y 422.468,Z 937.16,A -85,B 0,C 180,E1 7401.171,E2 7401.171} C_VEL
LIN {X 0,Y 429.329,Z 915.621,A -85,B 0,C 180,E1 7400.29,E2 7400.29} C_VEL
LIN {X 0,Y 436.854,Z 887.57,A -85,B 0,C 180,E1 7399.368,E2 7399.368} C_VEL
LIN {X 0,Y 441.795,Z 864.752,A -85,B 0,C 180,E1 7398.785,E2 7398.785} C_VEL
LIN {X 0,Y 445.607,Z 842.738,A -85,B 0,C 180,E1 7398.336,E2 7398.336} C_VEL
LIN {X 0,Y 448.918,Z 815.797,A -85,B 0,C 180,E1 7397.869,E2 7397.869} C_VEL
LIN {X 0,Y 469.503,Z 590.311,A -85,B 0,C 180,E1 7394.392,E2 7394.392} C_VEL
LIN {X 0,Y 470.835,Z 575.95,A -85,B 0,C 180,E1 7394.17,E2 7394.17} C_VEL
LIN {X 0,Y 466.137,Z 567.335,A -85,B 0,C 180,E1 7391.507,E2 7391.507} C_VEL
LIN {X 0,Y 462.647,Z 561.562,A -85,B 0,C 180,E1 7389.14,E2 7389.14} C_VEL
LIN {X 0,Y 460.838,Z 558.479,A -85,B 0,C 180,E1 7387.668,E2 7387.668} C_VEL
LIN {X 0,Y 458.871,Z 555.213,A -85,B 0,C 180,E1 7385.753,E2 7385.753} C_VEL
LIN {X 0,Y 456.444,Z 551.223,A -85,B 0,C 180,E1 7382.385,E2 7382.385} C_VEL
LIN {X 0,Y 455.188,Z 550.264,A -85,B 0,C 180,E1 7378.364,E2 7378.364} C_VEL
LIN {X 0,Y 455.505,Z 551.043,A -85,B 0,C 180,E1 7375.341,E2 7375.341} C_VEL
LIN {X 0,Y 457.494,Z 555.608,A -85,B 0,C 180,E1 7371.326,E2 7371.326} C_VEL
LIN {X 0,Y 459.543,Z 559.968,A -85,B 0,C 180,E1 7368.961,E2 7368.961} C_VEL
LIN {X 0,Y 461.711,Z 564.293,A -85,B 0,C 180,E1 7367.038,E2 7367.038} C_VEL
LIN {X 0,Y 464.891,Z 570.746,A -85,B 0,C 180,E1 7364.724,E2 7364.724} C_VEL
LIN {X 0,Y 468.949,Z 579.129,A -85,B 0,C 180,E1 7362.28,E2 7362.28} C_VEL
LIN {X 0,Y 469.121,Z 579.884,A -85,B 0,C 180,E1 7362.163,E2 7362.163} C_VEL
LIN {X 0,Y 449.118,Z 804.543,A -85,B 0,C 180,E1 7358.819,E2 7358.819} C_VEL
LIN {X 0,Y 445.442,Z 839.953,A -85,B 0,C 180,E1 7358.257,E2 7358.257} C_VEL
LIN {X 0,Y 441.531,Z 863.603,A -85,B 0,C 180,E1 7357.796,E2 7357.796} C_VEL
LIN {X 0,Y 436.892,Z 885.449,A -85,B 0,C 180,E1 7357.267,E2 7357.267} C_VEL
LIN {X 0,Y 430.43,Z 910.594,A -85,B 0,C 180,E1 7356.484,E2 7356.484} C_VEL
LIN {X 0,Y 422.907,Z 934.432,A -85,B 0,C 180,E1 7355.541,E2 7355.541} C_VEL
LIN {X 0,Y 416.054,Z 953.503,A -85,B 0,C 180,E1 7354.638,E2 7354.638} C_VEL
LIN {X 0,Y 407.823,Z 973.956,A -85,B 0,C 180,E1 7353.494,E2 7353.494} C_VEL
LIN {X 0,Y 396.526,Z 998.783,A -85,B 0,C 180,E1 7351.8,E2 7351.8} C_VEL
LIN {X 0,Y 386.984,Z 1017.597,A -85,B 0,C 180,E1 7350.244,E2 7350.244} C_VEL
LIN {X 0,Y 377.286,Z 1035.273,A -85,B 0,C 180,E1 7348.527,E2 7348.527} C_VEL
LIN {X 0,Y 364.944,Z 1056.006,A -85,B 0,C 180,E1 7346.116,E2 7346.116} C_VEL
LIN {X 0,Y 354.367,Z 1072.425,A -85,B 0,C 180,E1 7343.802,E2 7343.802} C_VEL
LIN {X 0,Y 344.533,Z 1086.939,A -85,B 0,C 180,E1 7341.394,E2 7341.394} C_VEL
LIN {X 0,Y 333.18,Z 1103.05,A -85,B 0,C 180,E1 7338.223,E2 7338.223} C_VEL
LIN {X 0,Y 322.472,Z 1117.429,A -85,B 0,C 180,E1 7334.737,E2 7334.737} C_VEL
LIN {X 0,Y 313.985,Z 1128.681,A -85,B 0,C 180,E1 7331.481,E2 7331.481} C_VEL
LIN {X 0,Y 305.725,Z 1139.652,A -85,B 0,C 180,E1 7327.705,E2 7327.705} C_VEL
LIN {X 0,Y 296.955,Z 1151.451,A -85,B 0,C 180,E1 7322.67,E2 7322.67} C_VEL
LIN {X 0,Y 291.373,Z 1159.331,A -85,B 0,C 180,E1 7318.49,E2 7318.49} C_VEL
LIN {X 0,Y 286.936,Z 1166.175,A -85,B 0,C 180,E1 7314.061,E2 7314.061} C_VEL
LIN {X 0,Y 283.093,Z 1173.018,A -85,B 0,C 180,E1 7308.322,E2 7308.322} C_VEL
LIN {X 0,Y 281.315,Z 1176.988,A -85,B 0,C 180,E1 7303.777,E2 7303.777} C_VEL
LIN {X 0,Y 280.447,Z 1179.717,A -85,B 0,C 180,E1 7299.44,E2 7299.44} C_VEL
LIN {X 0,Y 280.095,Z 1181.368,A -85,B 0,C 180,E1 7295.326,E2 7295.326} C_VEL
LIN {X 0,Y 280.018,Z 1182.109,A -85,B 0,C 180,E1 7291.228,E2 7291.228} C_VEL
LIN {X 0,Y 280.033,Z 1181.93,A -85,B 0,C 180,E1 7286.93,E2 7286.93} C_VEL
LIN {X 0,Y 280.276,Z 1180.535,A -85,B 0,C 180,E1 7282.003,E2 7282.003} C_VEL
LIN {X 0,Y 281.068,Z 1177.683,A -85,B 0,C 180,E1 7277.049,E2 7277.049} C_VEL
LIN {X 0,Y 282.558,Z 1174.114,A -85,B 0,C 180,E1 7272.708,E2 7272.708} C_VEL
LIN {X 0,Y 284.987,Z 1169.471,A -85,B 0,C 180,E1 7268.384,E2 7268.384} C_VEL
LIN {X 0,Y 289.324,Z 1162.548,A -85,B 0,C 180,E1 7263.304,E2 7263.304} C_VEL
LIN {X 0,Y 295.331,Z 1153.744,A -85,B 0,C 180,E1 7258.348,E2 7258.348} C_VEL
LIN {X 0,Y 301.74,Z 1144.998,A -85,B 0,C 180,E1 7254.324,E2 7254.324} C_VEL
LIN {X 0,Y 310.166,Z 1133.907,A -85,B 0,C 180,E1 7250.096,E2 7250.096} C_VEL
LIN {X 0,Y 320.003,Z 1120.844,A -85,B 0,C 180,E1 7246.08,E2 7246.08} C_VEL
LIN {X 0,Y 329.149,Z 1108.555,A -85,B 0,C 180,E1 7242.938,E2 7242.938} C_VEL
LIN {X 0,Y 339.169,Z 1094.757,A -85,B 0,C 180,E1 7239.961,E2 7239.961} C_VEL
LIN {X 0,Y 351.777,Z 1076.514,A -85,B 0,C 180,E1 7236.723,E2 7236.723} C_VEL
LIN {X 0,Y 362.207,Z 1060.482,A -85,B 0,C 180,E1 7234.372,E2 7234.372} C_VEL
LIN {X 0,Y 372.547,Z 1043.656,A -85,B 0,C 180,E1 7232.283,E2 7232.283} C_VEL
LIN {X 0,Y 385.406,Z 1020.875,A -85,B 0,C 180,E1 7229.945,E2 7229.945} C_VEL
LIN {X 0,Y 395.012,Z 1002.17,A -85,B 0,C 180,E1 7228.359,E2 7228.359} C_VEL
LIN {X 0,Y 403.597,Z 983.977,A -85,B 0,C 180,E1 7227.048,E2 7227.048} C_VEL
LIN {X 0,Y 413.622,Z 960.397,A -85,B 0,C 180,E1 7225.621,E2 7225.621} C_VEL
LIN {X 0,Y 414.63,Z 957.714,A -85,B 0,C 180,E1 7225.48,E2 7225.48} C_VEL
LIN {X 0,Y 416.769,Z 951.057,A -85,B 0,C 180,E1 7225.013,E2 7225.013} C_VEL
LIN {X 0,Y 420.628,Z 933.807,A -85,B 0,C 180,E1 7223.406,E2 7223.406} C_VEL
LIN {X 0,Y 422.317,Z 927.906,A -85,B 0,C 180,E1 7223.061,E2 7223.061} C_VEL
LIN {X 0,Y 429.529,Z 903.904,A -85,B 0,C 180,E1 7222.196,E2 7222.196} C_VEL
LIN {X 0,Y 434.822,Z 883.093,A -85,B 0,C 180,E1 7221.582,E2 7221.582} C_VEL
LIN {X 0,Y 439.506,Z 860.896,A -85,B 0,C 180,E1 7221.063,E2 7221.063} C_VEL
LIN {X 0,Y 443.947,Z 832.375,A -85,B 0,C 180,E1 7220.539,E2 7220.539} C_VEL
LIN {X 0,Y 449.539,Z 772.881,A -85,B 0,C 180,E1 7219.637,E2 7219.637} C_VEL
LIN {X 0,Y 466.716,Z 585.003,A -85,B 0,C 180,E1 7216.86,E2 7216.86} C_VEL
LIN {X 0,Y 462.64,Z 576.214,A -85,B 0,C 180,E1 7214.2,E2 7214.2} C_VEL
LIN {X 0,Y 459.182,Z 569.184,A -85,B 0,C 180,E1 7211.366,E2 7211.366} C_VEL
LIN {X 0,Y 457.152,Z 564.884,A -85,B 0,C 180,E1 7209.124,E2 7209.124} C_VEL
LIN {X 0,Y 456.077,Z 562.5,A -85,B 0,C 180,E1 7207.559,E2 7207.559} C_VEL
LIN {X 0,Y 454.621,Z 558.813,A -85,B 0,C 180,E1 7203.783,E2 7203.783} C_VEL
LIN {X 0,Y 454.749,Z 558.561,A -85,B 0,C 180,E1 7200,E2 7200} C_VEL
LIN {X 0,Y 455.836,Z 559.703,A -85,B 0,C 180,E1 7197.36,E2 7197.36} C_VEL
LIN {X 0,Y 458.552,Z 564.255,A -85,B 0,C 180,E1 7193.741,E2 7193.741} C_VEL
LIN {X 0,Y 461.067,Z 568.579,A -85,B 0,C 180,E1 7191.457,E2 7191.457} C_VEL
LIN {X 0,Y 464.638,Z 574.721,A -85,B 0,C 180,E1 7188.895,E2 7188.895} C_VEL
LIN {X 0,Y 468.313,Z 581.61,A -85,B 0,C 180,E1 7186.692,E2 7186.692} C_VEL
LIN {X 0,Y 447.191,Z 807.649,A -85,B 0,C 180,E1 7183.236,E2 7183.236} C_VEL
LIN {X 0,Y 443.42,Z 840.55,A -85,B 0,C 180,E1 7182.688,E2 7182.688} C_VEL
LIN {X 0,Y 439.515,Z 863.183,A -85,B 0,C 180,E1 7182.239,E2 7182.239} C_VEL
LIN {X 0,Y 434.902,Z 884.48,A -85,B 0,C 180,E1 7181.717,E2 7181.717} C_VEL
LIN {X 0,Y 428.415,Z 909.451,A -85,B 0,C 180,E1 7180.948,E2 7180.948} C_VEL
LIN {X 0,Y 420.387,Z 934.704,A -85,B 0,C 180,E1 7179.966,E2 7179.966} C_VEL
LIN {X 0,Y 412.957,Z 955.174,A -85,B 0,C 180,E1 7179.001,E2 7179.001} C_VEL
LIN {X 0,Y 404.754,Z 975.405,A -85,B 0,C 180,E1 7177.876,E2 7177.876} C_VEL
LIN {X 0,Y 394.164,Z 998.932,A -85,B 0,C 180,E1 7176.312,E2 7176.312} C_VEL
LIN {X 0,Y 383.137,Z 1020.676,A -85,B 0,C 180,E1 7174.549,E2 7174.549} C_VEL
LIN {X 0,Y 373.884,Z 1037.591,A -85,B 0,C 180,E1 7172.94,E2 7172.94} C_VEL
LIN {X 0,Y 364.082,Z 1054.349,A -85,B 0,C 180,E1 7171.095,E2 7171.095} C_VEL
LIN {X 0,Y 351.782,Z 1074.212,A -85,B 0,C 180,E1 7168.505,E2 7168.505} C_VEL
LIN {X 0,Y 340.045,Z 1091.781,A -85,B 0,C 180,E1 7165.716,E2 7165.716} C_VEL
LIN {X 0,Y 330.229,Z 1105.947,A -85,B 0,C 180,E1 7163.067,E2 7163.067} C_VEL
LIN {X 0,Y 320.605,Z 1119.472,A -85,B 0,C 180,E1 7160.103,E2 7160.103} C_VEL
LIN {X 0,Y 309.513,Z 1134.875,A -85,B 0,C 180,E1 7156.087,E2 7156.087} C_VEL
LIN {X 0,Y 299.799,Z 1148.079,A -85,B 0,C 180,E1 7151.838,E2 7151.838} C_VEL
LIN {X 0,Y 292.605,Z 1158.194,A -85,B 0,C 180,E1 7147.958,E2 7147.958} C_VEL
LIN {X 0,Y 286.289,Z 1167.494,A -85,B 0,C 180,E1 7143.732,E2 7143.732} C_VEL
LIN {X 0,Y 280.233,Z 1177.256,A -85,B 0,C 180,E1 7138.329,E2 7138.329} C_VEL
LIN {X 0,Y 276.245,Z 1184.577,A -85,B 0,C 180,E1 7133.165,E2 7133.165} C_VEL
LIN {X 0,Y 274.007,Z 1189.635,A -85,B 0,C 180,E1 7128.73,E2 7128.73} C_VEL
LIN {X 0,Y 272.743,Z 1193.495,A -85,B 0,C 180,E1 7124.435,E2 7124.435} C_VEL
LIN {X 0,Y 272.152,Z 1196.355,A -85,B 0,C 180,E1 7120.157,E2 7120.157} C_VEL
LIN {X 0,Y 271.995,Z 1198.083,A -85,B 0,C 180,E1 7116.331,E2 7116.331} C_VEL
LIN {X 0,Y 271.987,Z 1199.018,A -85,B 0,C 180,E1 7112.528,E2 7112.528} C_VEL
LIN {X 0,Y 271.993,Z 1199.161,A -85,B 0,C 180,E1 7108.736,E2 7108.736} C_VEL
LIN {X 0,Y 271.984,Z 1198.437,A -85,B 0,C 180,E1 7104.726,E2 7104.726} C_VEL
LIN {X 0,Y 272.105,Z 1196.704,A -85,B 0,C 180,E1 7100.482,E2 7100.482} C_VEL
LIN {X 0,Y 272.651,Z 1193.815,A -85,B 0,C 180,E1 7095.993,E2 7095.993} C_VEL
LIN {X 0,Y 273.847,Z 1190.034,A -85,B 0,C 180,E1 7091.684,E2 7091.684} C_VEL
LIN {X 0,Y 275.898,Z 1185.266,A -85,B 0,C 180,E1 7087.408,E2 7087.408} C_VEL
LIN {X 0,Y 279.096,Z 1179.121,A -85,B 0,C 180,E1 7082.936,E2 7082.936} C_VEL
LIN {X 0,Y 284.093,Z 1170.883,A -85,B 0,C 180,E1 7078.019,E2 7078.019} C_VEL
LIN {X 0,Y 291.464,Z 1159.815,A -85,B 0,C 180,E1 7072.74,E2 7072.74} C_VEL
LIN {X 0,Y 298.642,Z 1149.615,A -85,B 0,C 180,E1 7068.732,E2 7068.732} C_VEL
LIN {X 0,Y 306.378,Z 1138.94,A -85,B 0,C 180,E1 7065.176,E2 7065.176} C_VEL
LIN {X 0,Y 316.589,Z 1125.019,A -85,B 0,C 180,E1 7061.264,E2 7061.264} C_VEL
LIN {X 0,Y 328.115,Z 1108.866,A -85,B 0,C 180,E1 7057.552,E2 7057.552} C_VEL
LIN {X 0,Y 338.261,Z 1094.249,A -85,B 0,C 180,E1 7054.739,E2 7054.739} C_VEL
LIN {X 0,Y 348.335,Z 1079.211,A -85,B 0,C 180,E1 7052.27,E2 7052.27} C_VEL
LIN {X 0,Y 360.569,Z 1060.109,A -85,B 0,C 180,E1 7049.616,E2 7049.616} C_VEL
LIN {X 0,Y 372.474,Z 1039.86,A -85,B 0,C 180,E1 7047.309,E2 7047.309} C_VEL
LIN {X 0,Y 382.032,Z 1022.474,A -85,B 0,C 180,E1 7045.624,E2 7045.624} C_VEL
LIN {X 0,Y 391.528,Z 1003.884,A -85,B 0,C 180,E1 7044.079,E2 7044.079} C_VEL
LIN {X 0,Y 402.453,Z 980.555,A -85,B 0,C 180,E1 7042.449,E2 7042.449} C_VEL
LIN {X 0,Y 411.707,Z 958.027,A -85,B 0,C 180,E1 7041.158,E2 7041.158} C_VEL
LIN {X 0,Y 419.179,Z 937.715,A -85,B 0,C 180,E1 7040.177,E2 7040.177} C_VEL
LIN {X 0,Y 426.008,Z 916.741,A -85,B 0,C 180,E1 7039.326,E2 7039.326} C_VEL
LIN {X 0,Y 433.376,Z 890.318,A -85,B 0,C 180,E1 7038.453,E2 7038.453} C_VEL
LIN {X 0,Y 438.882,Z 865.516,A -85,B 0,C 180,E1 7037.82,E2 7037.82} C_VEL
LIN {X 0,Y 442.805,Z 843.361,A -85,B 0,C 180,E1 7037.372,E2 7037.372} C_VEL
LIN {X 0,Y 446.001,Z 818.192,A -85,B 0,C 180,E1 7036.939,E2 7036.939} C_VEL
LIN {X 0,Y 466.871,Z 594.698,A -85,B 0,C 180,E1 7033.513,E2 7033.513} C_VEL
LIN {X 0,Y 468.125,Z 581.374,A -85,B 0,C 180,E1 7033.306,E2 7033.306} C_VEL
LIN {X 0,Y 463.699,Z 573.324,A -85,B 0,C 180,E1 7030.624,E2 7030.624} C_VEL
LIN {X 0,Y 460.058,Z 566.902,A -85,B 0,C 180,E1 7027.87,E2 7027.87} C_VEL
LIN {X 0,Y 457.648,Z 562.943,A -85,B 0,C 180,E1 7025.517,E2 7025.517} C_VEL
LIN {X 0,Y 455.393,Z 559.121,A -85,B 0,C 180,E1 7022.265,E2 7022.265} C_VEL
LIN {X 0,Y 454.213,Z 558.204,A -85,B 0,C 180,E1 7018.36,E2 7018.36} C_VEL
LIN {X 0,Y 454.522,Z 559.074,A -85,B 0,C 180,E1 7015.331,E2 7015.331} C_VEL
LIN {X 0,Y 456.381,Z 563.418,A -85,B 0,C 180,E1 7011.495,E2 7011.495} C_VEL
LIN {X 0,Y 458.373,Z 567.798,A -85,B 0,C 180,E1 7009.124,E2 7009.124} C_VEL
LIN {X 0,Y 460.483,Z 572.131,A -85,B 0,C 180,E1 7007.204,E2 7007.204} C_VEL
LIN {X 0,Y 463.44,Z 578.312,A -85,B 0,C 180,E1 7004.995,E2 7004.995} C_VEL
LIN {X 0,Y 466.535,Z 584.875,A -85,B 0,C 180,E1 7003.039,E2 7003.039} C_VEL
LIN {X 0,Y 446.093,Z 809.484,A -85,B 0,C 180,E1 6999.718,E2 6999.718} C_VEL
LIN {X 0,Y 442.43,Z 842.202,A -85,B 0,C 180,E1 6999.193,E2 6999.193} C_VEL
LIN {X 0,Y 438.589,Z 864.678,A -85,B 0,C 180,E1 6998.756,E2 6998.756} C_VEL
LIN {X 0,Y 433.62,Z 887.445,A -85,B 0,C 180,E1 6998.206,E2 6998.206} C_VEL
LIN {X 0,Y 426.324,Z 914.37,A -85,B 0,C 180,E1 6997.354,E2 6997.354} C_VEL
LIN {X 0,Y 419.658,Z 935.001,A -85,B 0,C 180,E1 6996.535,E2 6996.535} C_VEL
LIN {X 0,Y 412.68,Z 954.014,A -85,B 0,C 180,E1 6995.645,E2 6995.645} C_VEL
LIN {X 0,Y 404.252,Z 974.527,A -85,B 0,C 180,E1 6994.508,E2 6994.508} C_VEL
LIN {X 0,Y 392.771,Z 999.181,A -85,B 0,C 180,E1 6992.839,E2 6992.839} C_VEL
LIN {X 0,Y 383.384,Z 1017.312,A -85,B 0,C 180,E1 6991.355,E2 6991.355} C_VEL
LIN {X 0,Y 373.669,Z 1034.647,A -85,B 0,C 180,E1 6989.692,E2 6989.692} C_VEL
LIN {X 0,Y 361.784,Z 1054.331,A -85,B 0,C 180,E1 6987.452,E2 6987.452} C_VEL
LIN {X 0,Y 349.808,Z 1072.422,A -85,B 0,C 180,E1 6984.933,E2 6984.933} C_VEL
LIN {X 0,Y 339.902,Z 1086.632,A -85,B 0,C 180,E1 6982.585,E2 6982.585} C_VEL
LIN {X 0,Y 328.986,Z 1101.624,A -85,B 0,C 180,E1 6979.656,E2 6979.656} C_VEL
LIN {X 0,Y 317.151,Z 1117.087,A -85,B 0,C 180,E1 6975.957,E2 6975.957} C_VEL
LIN {X 0,Y 307.816,Z 1128.986,A -85,B 0,C 180,E1 6972.492,E2 6972.492} C_VEL
LIN {X 0,Y 299.225,Z 1139.923,A -85,B 0,C 180,E1 6968.673,E2 6968.673} C_VEL
LIN {X 0,Y 290.24,Z 1151.445,A -85,B 0,C 180,E1 6963.687,E2 6963.687} C_VEL
LIN {X 0,Y 284.152,Z 1159.593,A -85,B 0,C 180,E1 6959.283,E2 6959.283} C_VEL
LIN {X 0,Y 279.447,Z 1166.435,A -85,B 0,C 180,E1 6954.749,E2 6954.749} C_VEL
LIN {X 0,Y 275.348,Z 1173.272,A -85,B 0,C 180,E1 6948.856,E2 6948.856} C_VEL
LIN {X 0,Y 273.436,Z 1177.24,A -85,B 0,C 180,E1 6944.182,E2 6944.182} C_VEL
LIN {X 0,Y 272.518,Z 1179.859,A -85,B 0,C 180,E1 6939.93,E2 6939.93} C_VEL
LIN {X 0,Y 272.116,Z 1181.552,A -85,B 0,C 180,E1 6935.694,E2 6935.694} C_VEL
LIN {X 0,Y 272.021,Z 1182.313,A -85,B 0,C 180,E1 6931.686,E2 6931.686} C_VEL
LIN {X 0,Y 272.029,Z 1182.282,A -85,B 0,C 180,E1 6927.894,E2 6927.894} C_VEL
LIN {X 0,Y 272.135,Z 1181.46,A -85,B 0,C 180,E1 6923.884,E2 6923.884} C_VEL
LIN {X 0,Y 272.533,Z 1179.813,A -85,B 0,C 180,E1 6919.858,E2 6919.858} C_VEL
LIN {X 0,Y 273.542,Z 1177.022,A -85,B 0,C 180,E1 6915.392,E2 6915.392} C_VEL
LIN {X 0,Y 275.888,Z 1172.393,A -85,B 0,C 180,E1 6910.082,E2 6910.082} C_VEL
LIN {X 0,Y 279.888,Z 1165.785,A -85,B 0,C 180,E1 6904.667,E2 6904.667} C_VEL
LIN {X 0,Y 284.554,Z 1159.096,A -85,B 0,C 180,E1 6900.301,E2 6900.301} C_VEL
LIN {X 0,Y 291.382,Z 1150.084,A -85,B 0,C 180,E1 6895.515,E2 6895.515} C_VEL
LIN {X 0,Y 300.243,Z 1138.678,A -85,B 0,C 180,E1 6890.748,E2 6890.748} C_VEL
LIN {X 0,Y 308.774,Z 1127.871,A -85,B 0,C 180,E1 6887.042,E2 6887.042} C_VEL
LIN {X 0,Y 319.493,Z 1114.297,A -85,B 0,C 180,E1 6883.182,E2 6883.182} C_VEL
LIN {X 0,Y 331.14,Z 1098.815,A -85,B 0,C 180,E1 6879.649,E2 6879.649} C_VEL
LIN {X 0,Y 340.906,Z 1085.386,A -85,B 0,C 180,E1 6877.083,E2 6877.083} C_VEL
LIN {X 0,Y 351.928,Z 1069.543,A -85,B 0,C 180,E1 6874.52,E2 6874.52} C_VEL
LIN {X 0,Y 364.907,Z 1049.444,A -85,B 0,C 180,E1 6871.851,E2 6871.851} C_VEL
LIN {X 0,Y 374.772,Z 1032.997,A -85,B 0,C 180,E1 6870.033,E2 6870.033} C_VEL
LIN {X 0,Y 384.272,Z 1015.971,A -85,B 0,C 180,E1 6868.422,E2 6868.422} C_VEL
LIN {X 0,Y 395.543,Z 994.015,A -85,B 0,C 180,E1 6866.672,E2 6866.672} C_VEL
LIN {X 0,Y 405.622,Z 971.691,A -85,B 0,C 180,E1 6865.222,E2 6865.222} C_VEL
LIN {X 0,Y 413.648,Z 951.946,A -85,B 0,C 180,E1 6864.148,E2 6864.148} C_VEL
LIN {X 0,Y 421.831,Z 929.309,A -85,B 0,C 180,E1 6863.12,E2 6863.12} C_VEL
LIN {X 0,Y 422.317,Z 927.906,A -85,B 0,C 180,E1 6863.061,E2 6863.061} C_VEL
LIN {X 0,Y 424.185,Z 920.961,A -85,B 0,C 180,E1 6862.662,E2 6862.662} C_VEL
LIN {X 0,Y 427.342,Z 902.811,A -85,B 0,C 180,E1 6861.245,E2 6861.245} C_VEL
LIN {X 0,Y 428.76,Z 896.692,A -85,B 0,C 180,E1 6860.956,E2 6860.956} C_VEL
LIN {X 0,Y 435.31,Z 869.089,A -85,B 0,C 180,E1 6860.246,E2 6860.246} C_VEL
LIN {X 0,Y 439.44,Z 846.319,A -85,B 0,C 180,E1 6859.793,E2 6859.793} C_VEL
LIN {X 0,Y 442.387,Z 823.898,A -85,B 0,C 180,E1 6859.419,E2 6859.419} C_VEL
LIN {X 0,Y 463.727,Z 595.625,A -85,B 0,C 180,E1 6856.064,E2 6856.064} C_VEL
LIN {X 0,Y 464.201,Z 590.36,A -85,B 0,C 180,E1 6855.972,E2 6855.972} C_VEL
LIN {X 0,Y 460.191,Z 581.582,A -85,B 0,C 180,E1 6853.124,E2 6853.124} C_VEL
LIN {X 0,Y 457.692,Z 576.391,A -85,B 0,C 180,E1 6850.893,E2 6850.893} C_VEL
LIN {X 0,Y 455.891,Z 572.38,A -85,B 0,C 180,E1 6848.768,E2 6848.768} C_VEL
LIN {X 0,Y 455.022,Z 570.382,A -85,B 0,C 180,E1 6847.449,E2 6847.449} C_VEL
LIN {X 0,Y 453.647,Z 566.76,A -85,B 0,C 180,E1 6843.791,E2 6843.791} C_VEL
LIN {X 0,Y 453.768,Z 566.503,A -85,B 0,C 180,E1 6840,E2 6840} C_VEL
LIN {X 0,Y 454.784,Z 567.581,A -85,B 0,C 180,E1 6837.48,E2 6837.48} C_VEL
LIN {X 0,Y 457.38,Z 572.053,A -85,B 0,C 180,E1 6833.914,E2 6833.914} C_VEL
LIN {X 0,Y 459.758,Z 576.259,A -85,B 0,C 180,E1 6831.684,E2 6831.684} C_VEL
LIN {X 0,Y 463.251,Z 582.404,A -85,B 0,C 180,E1 6829.114,E2 6829.114} C_VEL
LIN {X 0,Y 465.699,Z 587.307,A -85,B 0,C 180,E1 6827.558,E2 6827.558} C_VEL
LIN {X 0,Y 444.16,Z 813.374,A -85,B 0,C 180,E1 6824.128,E2 6824.128} C_VEL
LIN {X 0,Y 440.668,Z 841.739,A -85,B 0,C 180,E1 6823.652,E2 6823.652} C_VEL
LIN {X 0,Y 436.741,Z 863.951,A -85,B 0,C 180,E1 6823.215,E2 6823.215} C_VEL
LIN {X 0,Y 431.923,Z 885.69,A -85,B 0,C 180,E1 6822.687,E2 6822.687} C_VEL
LIN {X 0,Y 424.999,Z 911.529,A -85,B 0,C 180,E1 6821.891,E2 6821.891} C_VEL
LIN {X 0,Y 417.088,Z 935.724,A -85,B 0,C 180,E1 6820.953,E2 6820.953} C_VEL
LIN {X 0,Y 409.621,Z 955.841,A -85,B 0,C 180,E1 6820.013,E2 6820.013} C_VEL
LIN {X 0,Y 400.941,Z 976.76,A -85,B 0,C 180,E1 6818.857,E2 6818.857} C_VEL
LIN {X 0,Y 388.999,Z 1002.259,A -85,B 0,C 180,E1 6817.143,E2 6817.143} C_VEL
LIN {X 0,Y 379.179,Z 1021.147,A -85,B 0,C 180,E1 6815.607,E2 6815.607} C_VEL
LIN {X 0,Y 369.747,Z 1037.952,A -85,B 0,C 180,E1 6814.018,E2 6814.018} C_VEL
LIN {X 0,Y 359.493,Z 1055.016,A -85,B 0,C 180,E1 6812.142,E2 6812.142} C_VEL
LIN {X 0,Y 346.155,Z 1075.792,A -85,B 0,C 180,E1 6809.403,E2 6809.403} C_VEL
LIN {X 0,Y 334.754,Z 1092.341,A -85,B 0,C 180,E1 6806.754,E2 6806.754} C_VEL
LIN {X 0,Y 324.647,Z 1106.436,A -85,B 0,C 180,E1 6804.096,E2 6804.096} C_VEL
LIN {X 0,Y 314.185,Z 1120.624,A -85,B 0,C 180,E1 6800.94,E2 6800.94} C_VEL
LIN {X 0,Y 301.827,Z 1136.958,A -85,B 0,C 180,E1 6796.509,E2 6796.509} C_VEL
LIN {X 0,Y 292.74,Z 1148.866,A -85,B 0,C 180,E1 6792.553,E2 6792.553} C_VEL
LIN {X 0,Y 285.299,Z 1158.872,A -85,B 0,C 180,E1 6788.596,E2 6788.596} C_VEL
LIN {X 0,Y 277.661,Z 1169.732,A -85,B 0,C 180,E1 6783.433,E2 6783.433} C_VEL
LIN {X 0,Y 271.811,Z 1178.684,A -85,B 0,C 180,E1 6778.009,E2 6778.009} C_VEL
LIN {X 0,Y 268.386,Z 1184.767,A -85,B 0,C 180,E1 6773.492,E2 6773.492} C_VEL
LIN {X 0,Y 266.121,Z 1189.596,A -85,B 0,C 180,E1 6769.079,E2 6769.079} C_VEL
LIN {X 0,Y 264.784,Z 1193.41,A -85,B 0,C 180,E1 6764.655,E2 6764.655} C_VEL
LIN {X 0,Y 264.155,Z 1196.245,A -85,B 0,C 180,E1 6760.209,E2 6760.209} C_VEL
LIN {X 0,Y 263.993,Z 1197.979,A -85,B 0,C 180,E1 6756.087,E2 6756.087} C_VEL
LIN {X 0,Y 263.991,Z 1198.82,A -85,B 0,C 180,E1 6752.17,E2 6752.17} C_VEL
LIN {X 0,Y 263.996,Z 1198.89,A -85,B 0,C 180,E1 6748.48,E2 6748.48} C_VEL
LIN {X 0,Y 263.988,Z 1198.116,A -85,B 0,C 180,E1 6744.348,E2 6744.348} C_VEL
LIN {X 0,Y 264.123,Z 1196.453,A -85,B 0,C 180,E1 6740.191,E2 6740.191} C_VEL
LIN {X 0,Y 264.735,Z 1193.561,A -85,B 0,C 180,E1 6735.565,E2 6735.565} C_VEL
LIN {X 0,Y 266.031,Z 1189.791,A -85,B 0,C 180,E1 6731.141,E2 6731.141} C_VEL
LIN {X 0,Y 268.248,Z 1185.005,A -85,B 0,C 180,E1 6726.727,E2 6726.727} C_VEL
LIN {X 0,Y 271.681,Z 1178.857,A -85,B 0,C 180,E1 6722.134,E2 6722.134} C_VEL
LIN {X 0,Y 277.129,Z 1170.425,A -85,B 0,C 180,E1 6716.988,E2 6716.988} C_VEL
LIN {X 0,Y 284.959,Z 1159.292,A -85,B 0,C 180,E1 6711.605,E2 6711.605} C_VEL
LIN {X 0,Y 292.371,Z 1149.289,A -85,B 0,C 180,E1 6707.622,E2 6707.622} C_VEL
LIN {X 0,Y 300.896,Z 1138.066,A -85,B 0,C 180,E1 6703.855,E2 6703.855} C_VEL
LIN {X 0,Y 312.112,Z 1123.395,A -85,B 0,C 180,E1 6699.748,E2 6699.748} C_VEL
LIN {X 0,Y 323.774,Z 1107.519,A -85,B 0,C 180,E1 6696.147,E2 6696.147} C_VEL
LIN {X 0,Y 334.131,Z 1093.072,A -85,B 0,C 180,E1 6693.394,E2 6693.394} C_VEL
LIN {X 0,Y 345.492,Z 1076.587,A -85,B 0,C 180,E1 6690.735,E2 6690.735} C_VEL
LIN {X 0,Y 358.88,Z 1055.817,A -85,B 0,C 180,E1 6687.969,E2 6687.969} C_VEL
LIN {X 0,Y 369.656,Z 1037.865,A -85,B 0,C 180,E1 6685.989,E2 6685.989} C_VEL
LIN {X 0,Y 379.08,Z 1021.051,A -85,B 0,C 180,E1 6684.4,E2 6684.4} C_VEL
LIN {X 0,Y 389.366,Z 1001.236,A -85,B 0,C 180,E1 6682.794,E2 6682.794} C_VEL
LIN {X 0,Y 400.924,Z 976.422,A -85,B 0,C 180,E1 6681.135,E2 6681.135} C_VEL
LIN {X 0,Y 409.535,Z 955.641,A -85,B 0,C 180,E1 6679.988,E2 6679.988} C_VEL
LIN {X 0,Y 416.825,Z 935.987,A -85,B 0,C 180,E1 6679.069,E2 6679.069} C_VEL
LIN {X 0,Y 424.57,Z 912.321,A -85,B 0,C 180,E1 6678.147,E2 6678.147} C_VEL
LIN {X 0,Y 431.75,Z 885.664,A -85,B 0,C 180,E1 6677.322,E2 6677.322} C_VEL
LIN {X 0,Y 436.566,Z 863.917,A -85,B 0,C 180,E1 6676.792,E2 6676.792} C_VEL
LIN {X 0,Y 440.516,Z 841.531,A -85,B 0,C 180,E1 6676.352,E2 6676.352} C_VEL
LIN {X 0,Y 444.103,Z 811.983,A -85,B 0,C 180,E1 6675.859,E2 6675.859} C_VEL
LIN {X 0,Y 465.511,Z 587.136,A -85,B 0,C 180,E1 6672.446,E2 6672.446} C_VEL
LIN {X 0,Y 462.322,Z 581.012,A -85,B 0,C 180,E1 6670.404,E2 6670.404} C_VEL
LIN {X 0,Y 458.771,Z 574.59,A -85,B 0,C 180,E1 6667.64,E2 6667.64} C_VEL
LIN {X 0,Y 456.544,Z 570.816,A -85,B 0,C 180,E1 6665.404,E2 6665.404} C_VEL
LIN {X 0,Y 454.344,Z 567.02,A -85,B 0,C 180,E1 6662.144,E2 6662.144} C_VEL
LIN {X 0,Y 453.233,Z 566.145,A -85,B 0,C 180,E1 6658.357,E2 6658.357} C_VEL
LIN {X 0,Y 453.514,Z 566.959,A -85,B 0,C 180,E1 6655.448,E2 6655.448} C_VEL
LIN {X 0,Y 455.314,Z 571.336,A -85,B 0,C 180,E1 6651.603,E2 6651.603} C_VEL
LIN {X 0,Y 457.206,Z 575.626,A -85,B 0,C 180,E1 6649.287,E2 6649.287} C_VEL
LIN {X 0,Y 459.494,Z 580.436,A -85,B 0,C 180,E1 6647.176,E2 6647.176} C_VEL
LIN {X 0,Y 462.898,Z 587.721,A -85,B 0,C 180,E1 6644.656,E2 6644.656} C_VEL
LIN {X 0,Y 464.006,Z 590.469,A -85,B 0,C 180,E1 6643.915,E2 6643.915} C_VEL
LIN {X 0,Y 442.995,Z 816.439,A -85,B 0,C 180,E1 6640.599,E2 6640.599} C_VEL
LIN {X 0,Y 439.653,Z 843.699,A -85,B 0,C 180,E1 6640.155,E2 6640.155} C_VEL
LIN {X 0,Y 435.811,Z 865.551,A -85,B 0,C 180,E1 6639.732,E2 6639.732} C_VEL
LIN {X 0,Y 430.339,Z 889.99,A -85,B 0,C 180,E1 6639.143,E2 6639.143} C_VEL
LIN {X 0,Y 423.315,Z 915.013,A -85,B 0,C 180,E1 6638.35,E2 6638.35} C_VEL
LIN {X 0,Y 416.537,Z 935.569,A -85,B 0,C 180,E1 6637.545,E2 6637.545} C_VEL
LIN {X 0,Y 409.436,Z 954.524,A -85,B 0,C 180,E1 6636.668,E2 6636.668} C_VEL
LIN {X 0,Y 400.137,Z 976.664,A -85,B 0,C 180,E1 6635.447,E2 6635.447} C_VEL
LIN {X 0,Y 389.149,Z 999.575,A -85,B 0,C 180,E1 6633.897,E2 6633.897} C_VEL
LIN {X 0,Y 379.568,Z 1017.683,A -85,B 0,C 180,E1 6632.428,E2 6632.428} C_VEL
LIN {X 0,Y 369.892,Z 1034.563,A -85,B 0,C 180,E1 6630.824,E2 6630.824} C_VEL
LIN {X 0,Y 357.802,Z 1054.147,A -85,B 0,C 180,E1 6628.619,E2 6628.619} C_VEL
LIN {X 0,Y 345.591,Z 1072.131,A -85,B 0,C 180,E1 6626.136,E2 6626.136} C_VEL
LIN {X 0,Y 335.561,Z 1086.13,A -85,B 0,C 180,E1 6623.843,E2 6623.843} C_VEL
LIN {X 0,Y 324.974,Z 1100.235,A -85,B 0,C 180,E1 6621.117,E2 6621.117} C_VEL
LIN {X 0,Y 311.983,Z 1116.743,A -85,B 0,C 180,E1 6617.217,E2 6617.217} C_VEL
LIN {X 0,Y 302.255,Z 1128.67,A -85,B 0,C 180,E1 6613.74,E2 6613.74} C_VEL
LIN {X 0,Y 293.61,Z 1139.193,A -85,B 0,C 180,E1 6610.064,E2 6610.064} C_VEL
LIN {X 0,Y 284.389,Z 1150.533,A -85,B 0,C 180,E1 6605.213,E2 6605.213} C_VEL
LIN {X 0,Y 277.513,Z 1159.171,A -85,B 0,C 180,E1 6600.533,E2 6600.533} C_VEL
LIN {X 0,Y 272.592,Z 1165.818,A -85,B 0,C 180,E1 6596.115,E2 6596.115} C_VEL
LIN {X 0,Y 268.523,Z 1172.044,A -85,B 0,C 180,E1 6590.945,E2 6590.945} C_VEL
LIN {X 0,Y 265.784,Z 1177.037,A -85,B 0,C 180,E1 6585.269,E2 6585.269} C_VEL
LIN {X 0,Y 264.599,Z 1180.002,A -85,B 0,C 180,E1 6580.451,E2 6580.451} C_VEL
LIN {X 0,Y 264.154,Z 1181.671,A -85,B 0,C 180,E1 6576.303,E2 6576.303} C_VEL
LIN {X 0,Y 264.031,Z 1182.518,A -85,B 0,C 180,E1 6572.171,E2 6572.171} C_VEL
LIN {X 0,Y 264.031,Z 1182.572,A -85,B 0,C 180,E1 6568.264,E2 6568.264} C_VEL
LIN {X 0,Y 264.127,Z 1181.836,A -85,B 0,C 180,E1 6564.134,E2 6564.134} C_VEL
LIN {X 0,Y 264.518,Z 1180.278,A -85,B 0,C 180,E1 6559.987,E2 6559.987} C_VEL
LIN {X 0,Y 265.472,Z 1177.729,A -85,B 0,C 180,E1 6555.607,E2 6555.607} C_VEL
LIN {X 0,Y 267.345,Z 1174.027,A -85,B 0,C 180,E1 6551.012,E2 6551.012} C_VEL
LIN {X 0,Y 271.179,Z 1168.015,A -85,B 0,C 180,E1 6545.377,E2 6545.377} C_VEL
LIN {X 0,Y 276.633,Z 1160.378,A -85,B 0,C 180,E1 6540.08,E2 6540.08} C_VEL
LIN {X 0,Y 282.642,Z 1152.698,A -85,B 0,C 180,E1 6535.773,E2 6535.773} C_VEL
LIN {X 0,Y 291.114,Z 1142.405,A -85,B 0,C 180,E1 6531.058,E2 6531.058} C_VEL
LIN {X 0,Y 301.196,Z 1130.066,A -85,B 0,C 180,E1 6526.594,E2 6526.594} C_VEL
LIN {X 0,Y 310.296,Z 1118.914,A -85,B 0,C 180,E1 6523.261,E2 6523.261} C_VEL
LIN {X 0,Y 321.433,Z 1105.001,A -85,B 0,C 180,E1 6519.796,E2 6519.796} C_VEL
LIN {X 0,Y 334.198,Z 1088.166,A -85,B 0,C 180,E1 6516.408,E2 6516.408} C_VEL
LIN {X 0,Y 344.771,Z 1073.482,A -85,B 0,C 180,E1 6513.96,E2 6513.96} C_VEL
LIN {X 0,Y 355.921,Z 1057.12,A -85,B 0,C 180,E1 6511.657,E2 6511.657} C_VEL
LIN {X 0,Y 369.006,Z 1036.332,A -85,B 0,C 180,E1 6509.249,E2 6509.249} C_VEL
LIN {X 0,Y 379.385,Z 1018.309,A -85,B 0,C 180,E1 6507.52,E2 6507.52} C_VEL
LIN {X 0,Y 388.967,Z 1000.261,A -85,B 0,C 180,E1 6506.049,E2 6506.049} C_VEL
LIN {X 0,Y 399.963,Z 977.484,A -85,B 0,C 180,E1 6504.499,E2 6504.499} C_VEL
LIN {X 0,Y 409.26,Z 955.426,A -85,B 0,C 180,E1 6503.276,E2 6503.276} C_VEL
LIN {X 0,Y 416.359,Z 936.581,A -85,B 0,C 180,E1 6502.397,E2 6502.397} C_VEL
LIN {X 0,Y 423.218,Z 915.905,A -85,B 0,C 180,E1 6501.581,E2 6501.581} C_VEL
LIN {X 0,Y 428.76,Z 896.692,A -85,B 0,C 180,E1 6500.956,E2 6500.956} C_VEL
LIN {X 0,Y 430.18,Z 890.518,A -85,B 0,C 180,E1 6500.679,E2 6500.679} C_VEL
LIN {X 0,Y 432.628,Z 871.681,A -85,B 0,C 180,E1 6499.418,E2 6499.418} C_VEL
LIN {X 0,Y 433.775,Z 864.33,A -85,B 0,C 180,E1 6499.135,E2 6499.135} C_VEL
LIN {X 0,Y 437.768,Z 841.634,A -85,B 0,C 180,E1 6498.71,E2 6498.71} C_VEL
LIN {X 0,Y 441.728,Z 806.955,A -85,B 0,C 180,E1 6498.168,E2 6498.168} C_VEL
LIN {X 0,Y 461.81,Z 595.879,A -85,B 0,C 180,E1 6495.095,E2 6495.095} C_VEL
LIN {X 0,Y 458.525,Z 588.518,A -85,B 0,C 180,E1 6492.596,E2 6492.596} C_VEL
LIN {X 0,Y 456.292,Z 583.711,A -85,B 0,C 180,E1 6490.479,E2 6490.479} C_VEL
LIN {X 0,Y 454.64,Z 579.871,A -85,B 0,C 180,E1 6488.41,E2 6488.41} C_VEL
LIN {X 0,Y 453.892,Z 578.146,A -85,B 0,C 180,E1 6487.214,E2 6487.214} C_VEL
LIN {X 0,Y 452.649,Z 574.671,A -85,B 0,C 180,E1 6483.673,E2 6483.673} C_VEL
LIN {X 0,Y 452.788,Z 574.445,A -85,B 0,C 180,E1 6480,E2 6480} C_VEL
LIN {X 0,Y 453.734,Z 575.459,A -85,B 0,C 180,E1 6477.6,E2 6477.6} C_VEL
LIN {X 0,Y 456.213,Z 579.85,A -85,B 0,C 180,E1 6474.087,E2 6474.087} C_VEL
LIN {X 0,Y 458.461,Z 583.94,A -85,B 0,C 180,E1 6471.913,E2 6471.913} C_VEL
LIN {X 0,Y 461.779,Z 589.938,A -85,B 0,C 180,E1 6469.394,E2 6469.394} C_VEL
LIN {X 0,Y 463.187,Z 593.049,A -85,B 0,C 180,E1 6468.434,E2 6468.434} C_VEL
LIN {X 0,Y 441.312,Z 817.895,A -85,B 0,C 180,E1 6465.049,E2 6465.049} C_VEL
LIN {X 0,Y 438,Z 843.195,A -85,B 0,C 180,E1 6464.623,E2 6464.623} C_VEL
LIN {X 0,Y 434.011,Z 865.139,A -85,B 0,C 180,E1 6464.195,E2 6464.195} C_VEL
LIN {X 0,Y 428.634,Z 888.717,A -85,B 0,C 180,E1 6463.622,E2 6463.622} C_VEL
LIN {X 0,Y 421.276,Z 914.776,A -85,B 0,C 180,E1 6462.806,E2 6462.806} C_VEL
LIN {X 0,Y 413.825,Z 936.994,A -85,B 0,C 180,E1 6461.946,E2 6461.946} C_VEL
LIN {X 0,Y 406.076,Z 957.364,A -85,B 0,C 180,E1 6460.999,E2 6460.999} C_VEL
LIN {X 0,Y 396.063,Z 980.853,A -85,B 0,C 180,E1 6459.695,E2 6459.695} C_VEL
LIN {X 0,Y 384.694,Z 1004.096,A -85,B 0,C 180,E1 6458.108,E2 6458.108} C_VEL
LIN {X 0,Y 375.26,Z 1021.784,A -85,B 0,C 180,E1 6456.672,E2 6456.672} C_VEL
LIN {X 0,Y 365.563,Z 1038.619,A -85,B 0,C 180,E1 6455.088,E2 6455.088} C_VEL
LIN {X 0,Y 353.382,Z 1058.35,A -85,B 0,C 180,E1 6452.9,E2 6452.9} C_VEL
LIN {X 0,Y 339.952,Z 1078.314,A -85,B 0,C 180,E1 6450.187,E2 6450.187} C_VEL
LIN {X 0,Y 328.839,Z 1093.919,A -85,B 0,C 180,E1 6447.645,E2 6447.645} C_VEL
LIN {X 0,Y 317.423,Z 1109.298,A -85,B 0,C 180,E1 6444.67,E2 6444.67} C_VEL
LIN {X 0,Y 304.117,Z 1126.495,A -85,B 0,C 180,E1 6440.59,E2 6440.59} C_VEL
LIN {X 0,Y 294.154,Z 1139.042,A -85,B 0,C 180,E1 6436.954,E2 6436.954} C_VEL
LIN {X 0,Y 285.315,Z 1150.184,A -85,B 0,C 180,E1 6433.107,E2 6433.107} C_VEL
LIN {X 0,Y 275.967,Z 1162.332,A -85,B 0,C 180,E1 6428.02,E2 6428.02} C_VEL
LIN {X 0,Y 268.76,Z 1172.043,A -85,B 0,C 180,E1 6422.899,E2 6422.899} C_VEL
LIN {X 0,Y 263.91,Z 1179.263,A -85,B 0,C 180,E1 6418.267,E2 6418.267} C_VEL
LIN {X 0,Y 260.351,Z 1185.306,A -85,B 0,C 180,E1 6413.541,E2 6413.541} C_VEL
LIN {X 0,Y 257.65,Z 1191.076,A -85,B 0,C 180,E1 6407.853,E2 6407.853} C_VEL
LIN {X 0,Y 256.341,Z 1195.128,A -85,B 0,C 180,E1 6402.159,E2 6402.159} C_VEL
LIN {X 0,Y 256.025,Z 1197.367,A -85,B 0,C 180,E1 6397.404,E2 6397.404} C_VEL
LIN {X 0,Y 255.991,Z 1198.475,A -85,B 0,C 180,E1 6393.134,E2 6393.134} C_VEL
LIN {X 0,Y 255.999,Z 1198.69,A -85,B 0,C 180,E1 6388.881,E2 6388.881} C_VEL
LIN {X 0,Y 255.99,Z 1197.94,A -85,B 0,C 180,E1 6384.396,E2 6384.396} C_VEL
LIN {X 0,Y 256.146,Z 1196.201,A -85,B 0,C 180,E1 6379.883,E2 6379.883} C_VEL
LIN {X 0,Y 256.827,Z 1193.306,A -85,B 0,C 180,E1 6375.11,E2 6375.11} C_VEL
LIN {X 0,Y 258.245,Z 1189.533,A -85,B 0,C 180,E1 6370.55,E2 6370.55} C_VEL
LIN {X 0,Y 260.698,Z 1184.621,A -85,B 0,C 180,E1 6365.901,E2 6365.901} C_VEL
LIN {X 0,Y 264.313,Z 1178.593,A -85,B 0,C 180,E1 6361.286,E2 6361.286} C_VEL
LIN {X 0,Y 270.111,Z 1170.158,A -85,B 0,C 180,E1 6356.016,E2 6356.016} C_VEL
LIN {X 0,Y 278.38,Z 1159.016,A -85,B 0,C 180,E1 6350.524,E2 6350.524} C_VEL
LIN {X 0,Y 286.146,Z 1149.057,A -85,B 0,C 180,E1 6346.498,E2 6346.498} C_VEL
LIN {X 0,Y 294.624,Z 1138.373,A -85,B 0,C 180,E1 6342.857,E2 6342.857} C_VEL
LIN {X 0,Y 305.7,Z 1124.444,A -85,B 0,C 180,E1 6338.881,E2 6338.881} C_VEL
LIN {X 0,Y 318.202,Z 1108.103,A -85,B 0,C 180,E1 6335.103,E2 6335.103} C_VEL
LIN {X 0,Y 328.936,Z 1093.626,A -85,B 0,C 180,E1 6332.323,E2 6332.323} C_VEL
LIN {X 0,Y 339.939,Z 1078.158,A -85,B 0,C 180,E1 6329.807,E2 6329.807} C_VEL
LIN {X 0,Y 353.304,Z 1058.26,A -85,B 0,C 180,E1 6327.107,E2 6327.107} C_VEL
LIN {X 0,Y 365.116,Z 1039.128,A -85,B 0,C 180,E1 6324.98,E2 6324.98} C_VEL
LIN {X 0,Y 375.156,Z 1021.688,A -85,B 0,C 180,E1 6323.335,E2 6323.335} C_VEL
LIN {X 0,Y 385.068,Z 1003.062,A -85,B 0,C 180,E1 6321.829,E2 6321.829} C_VEL
LIN {X 0,Y 396.773,Z 978.827,A -85,B 0,C 180,E1 6320.197,E2 6320.197} C_VEL
LIN {X 0,Y 406.06,Z 956.974,A -85,B 0,C 180,E1 6318.992,E2 6318.992} C_VEL
LIN {X 0,Y 413.398,Z 937.69,A -85,B 0,C 180,E1 6318.095,E2 6318.095} C_VEL
LIN {X 0,Y 420.424,Z 916.853,A -85,B 0,C 180,E1 6317.278,E2 6317.278} C_VEL
LIN {X 0,Y 427.955,Z 890.784,A -85,B 0,C 180,E1 6316.443,E2 6316.443} C_VEL
LIN {X 0,Y 433.703,Z 865.726,A -85,B 0,C 180,E1 6315.826,E2 6315.826} C_VEL
LIN {X 0,Y 437.747,Z 843.577,A -85,B 0,C 180,E1 6315.392,E2 6315.392} C_VEL
LIN {X 0,Y 441.003,Z 818.884,A -85,B 0,C 180,E1 6314.975,E2 6314.975} C_VEL
LIN {X 0,Y 462.653,Z 596.306,A -85,B 0,C 180,E1 6311.621,E2 6311.621} C_VEL
LIN {X 0,Y 462.999,Z 592.586,A -85,B 0,C 180,E1 6311.555,E2 6311.555} C_VEL
LIN {X 0,Y 459.544,Z 586.075,A -85,B 0,C 180,E1 6309.139,E2 6309.139} C_VEL
LIN {X 0,Y 457.019,Z 581.535,A -85,B 0,C 180,E1 6306.974,E2 6306.974} C_VEL
LIN {X 0,Y 455.332,Z 578.546,A -85,B 0,C 180,E1 6305.166,E2 6305.166} C_VEL
LIN {X 0,Y 453.297,Z 574.918,A -85,B 0,C 180,E1 6302.023,E2 6302.023} C_VEL
LIN {X 0,Y 452.246,Z 574.093,A -85,B 0,C 180,E1 6298.226,E2 6298.226} C_VEL
LIN {X 0,Y 452.509,Z 574.844,A -85,B 0,C 180,E1 6295.564,E2 6295.564} C_VEL
LIN {X 0,Y 454.207,Z 579.146,A -85,B 0,C 180,E1 6291.773,E2 6291.773} C_VEL
LIN {X 0,Y 455.986,Z 583.323,A -85,B 0,C 180,E1 6289.513,E2 6289.513} C_VEL
LIN {X 0,Y 458.282,Z 588.287,A -85,B 0,C 180,E1 6287.334,E2 6287.334} C_VEL
LIN {X 0,Y 461.611,Z 595.738,A -85,B 0,C 180,E1 6284.805,E2 6284.805} C_VEL
LIN {X 0,Y 440.115,Z 821.347,A -85,B 0,C 180,E1 6281.519,E2 6281.519} C_VEL
LIN {X 0,Y 437.002,Z 845.197,A -85,B 0,C 180,E1 6281.129,E2 6281.129} C_VEL
LIN {X 0,Y 432.971,Z 867.389,A -85,B 0,C 180,E1 6280.7,E2 6280.7} C_VEL
LIN {X 0,Y 426.798,Z 893.771,A -85,B 0,C 180,E1 6280.056,E2 6280.056} C_VEL
LIN {X 0,Y 420.025,Z 916.928,A -85,B 0,C 180,E1 6279.317,E2 6279.317} C_VEL
LIN {X 0,Y 413.143,Z 937.256,A -85,B 0,C 180,E1 6278.522,E2 6278.522} C_VEL
LIN {X 0,Y 405.535,Z 957.022,A -85,B 0,C 180,E1 6277.607,E2 6277.607} C_VEL
LIN {X 0,Y 394.523,Z 982.084,A -85,B 0,C 180,E1 6276.194,E2 6276.194} C_VEL
LIN {X 0,Y 384.52,Z 1002.146,A -85,B 0,C 180,E1 6274.812,E2 6274.812} C_VEL
LIN {X 0,Y 374.771,Z 1020.029,A -85,B 0,C 180,E1 6273.351,E2 6273.351} C_VEL
LIN {X 0,Y 362.407,Z 1040.839,A -85,B 0,C 180,E1 6271.326,E2 6271.326} C_VEL
LIN {X 0,Y 350.157,Z 1059.454,A -85,B 0,C 180,E1 6269.102,E2 6269.102} C_VEL
LIN {X 0,Y 339.781,Z 1074.257,A -85,B 0,C 180,E1 6267.001,E2 6267.001} C_VEL
LIN {X 0,Y 328.55,Z 1089.406,A -85,B 0,C 180,E1 6264.459,E2 6264.459} C_VEL
LIN {X 0,Y 314.67,Z 1106.999,A -85,B 0,C 180,E1 6260.835,E2 6260.835} C_VEL
LIN {X 0,Y 304.28,Z 1119.561,A -85,B 0,C 180,E1 6257.651,E2 6257.651} C_VEL
LIN {X 0,Y 294.45,Z 1131.178,A -85,B 0,C 180,E1 6254.118,E2 6254.118} C_VEL
LIN {X 0,Y 283.248,Z 1144.227,A -85,B 0,C 180,E1 6249.189,E2 6249.189} C_VEL
LIN {X 0,Y 275.49,Z 1153.307,A -85,B 0,C 180,E1 6244.888,E2 6244.888} C_VEL
LIN {X 0,Y 269.073,Z 1161.137,A -85,B 0,C 180,E1 6240.357,E2 6240.357} C_VEL
LIN {X 0,Y 263.037,Z 1169.129,A -85,B 0,C 180,E1 6234.478,E2 6234.478} C_VEL
LIN {X 0,Y 259.505,Z 1174.445,A -85,B 0,C 180,E1 6229.264,E2 6229.264} C_VEL
LIN {X 0,Y 257.562,Z 1178.048,A -85,B 0,C 180,E1 6224.616,E2 6224.616} C_VEL
LIN {X 0,Y 256.52,Z 1180.682,A -85,B 0,C 180,E1 6219.876,E2 6219.876} C_VEL
LIN {X 0,Y 256.094,Z 1182.371,A -85,B 0,C 180,E1 6214.928,E2 6214.928} C_VEL
LIN {X 0,Y 256.032,Z 1182.981,A -85,B 0,C 180,E1 6210,E2 6210} C_VEL
LIN {X 0,Y 256.099,Z 1182.342,A -85,B 0,C 180,E1 6204.848,E2 6204.848} C_VEL
LIN {X 0,Y 256.505,Z 1180.742,A -85,B 0,C 180,E1 6200.125,E2 6200.125} C_VEL
LIN {X 0,Y 257.536,Z 1178.131,A -85,B 0,C 180,E1 6195.383,E2 6195.383} C_VEL
LIN {X 0,Y 259.505,Z 1174.478,A -85,B 0,C 180,E1 6190.649,E2 6190.649} C_VEL
LIN {X 0,Y 262.967,Z 1169.259,A -85,B 0,C 180,E1 6185.516,E2 6185.516} C_VEL
LIN {X 0,Y 269.072,Z 1161.198,A -85,B 0,C 180,E1 6179.557,E2 6179.557} C_VEL
LIN {X 0,Y 275.511,Z 1153.349,A -85,B 0,C 180,E1 6175.012,E2 6175.012} C_VEL
LIN {X 0,Y 283.63,Z 1143.876,A -85,B 0,C 180,E1 6170.538,E2 6170.538} C_VEL
LIN {X 0,Y 294.772,Z 1130.895,A -85,B 0,C 180,E1 6165.673,E2 6165.673} C_VEL
LIN {X 0,Y 304.696,Z 1119.186,A -85,B 0,C 180,E1 6162.13,E2 6162.13} C_VEL
LIN {X 0,Y 315.647,Z 1105.964,A -85,B 0,C 180,E1 6158.808,E2 6158.808} C_VEL
LIN {X 0,Y 328.767,Z 1089.288,A -85,B 0,C 180,E1 6155.407,E2 6155.407} C_VEL
LIN {X 0,Y 339.607,Z 1074.692,A -85,B 0,C 180,E1 6152.955,E2 6152.955} C_VEL
LIN {X 0,Y 350.323,Z 1059.426,A -85,B 0,C 180,E1 6150.785,E2 6150.785} C_VEL
LIN {X 0,Y 362.95,Z 1040.253,A -85,B 0,C 180,E1 6148.503,E2 6148.503} C_VEL
LIN {X 0,Y 374.85,Z 1020.192,A -85,B 0,C 180,E1 6146.557,E2 6146.557} C_VEL
LIN {X 0,Y 384.918,Z 1001.726,A -85,B 0,C 180,E1 6145.051,E2 6145.051} C_VEL
LIN {X 0,Y 395.129,Z 981.213,A -85,B 0,C 180,E1 6143.646,E2 6143.646} C_VEL
LIN {X 0,Y 405.76,Z 956.918,A -85,B 0,C 180,E1 6142.286,E2 6142.286} C_VEL
LIN {X 0,Y 413.376,Z 937.133,A -85,B 0,C 180,E1 6141.372,E2 6141.372} C_VEL
LIN {X 0,Y 420.414,Z 916.319,A -85,B 0,C 180,E1 6140.562,E2 6140.562} C_VEL
LIN {X 0,Y 427.868,Z 890.446,A -85,B 0,C 180,E1 6139.752,E2 6139.752} C_VEL
LIN {X 0,Y 433.502,Z 865.703,A -85,B 0,C 180,E1 6139.164,E2 6139.164} C_VEL
LIN {X 0,Y 433.775,Z 864.33,A -85,B 0,C 180,E1 6139.135,E2 6139.135} C_VEL
LIN {X 0,Y 435.002,Z 856.931,A -85,B 0,C 180,E1 6138.865,E2 6138.865} C_VEL
LIN {X 0,Y 436.362,Z 837.575,A -85,B 0,C 180,E1 6137.725,E2 6137.725} C_VEL
LIN {X 0,Y 436.959,Z 831.119,A -85,B 0,C 180,E1 6137.528,E2 6137.528} C_VEL
LIN {X 0,Y 444.285,Z 757.241,A -85,B 0,C 180,E1 6136.442,E2 6136.442} C_VEL
LIN {X 0,Y 459.501,Z 601.513,A -85,B 0,C 180,E1 6134.202,E2 6134.202} C_VEL
LIN {X 0,Y 456.893,Z 595.486,A -85,B 0,C 180,E1 6132.064,E2 6132.064} C_VEL
LIN {X 0,Y 454.863,Z 590.893,A -85,B 0,C 180,E1 6130.001,E2 6130.001} C_VEL
LIN {X 0,Y 453.074,Z 586.381,A -85,B 0,C 180,E1 6127.482,E2 6127.482} C_VEL
LIN {X 0,Y 451.653,Z 582.583,A -85,B 0,C 180,E1 6123.554,E2 6123.554} C_VEL
LIN {X 0,Y 451.84,Z 582.416,A -85,B 0,C 180,E1 6119.873,E2 6119.873} C_VEL
LIN {X 0,Y 452.686,Z 583.337,A -85,B 0,C 180,E1 6117.721,E2 6117.721} C_VEL
LIN {X 0,Y 455.104,Z 587.763,A -85,B 0,C 180,E1 6114.199,E2 6114.199} C_VEL
LIN {X 0,Y 457.243,Z 591.763,A -85,B 0,C 180,E1 6112.081,E2 6112.081} C_VEL
LIN {X 0,Y 460.4,Z 597.649,A -85,B 0,C 180,E1 6109.615,E2 6109.615} C_VEL
LIN {X 0,Y 460.797,Z 598.66,A -85,B 0,C 180,E1 6109.321,E2 6109.321} C_VEL
